VAR
	pGCodeTool		: POINTER TO FB_GCodeTool;
END_VAR
CASE eType OF
	E_PrintParamType.Pressure:
		CASE nNumerator OF
			1:	IF aiDispenser[1] <> 0 AND_THEN 
					(aiDispenser[1].P_pObject^.P_eObjectType = E_ObjectType.OBJECTTYPE_CartDispenser OR	aiDispenser[1].P_pObject^.P_eObjectType = E_ObjectType.OBJECTTYPE_CartDispStirrer) THEN
					pGCodeTool := aiDispenser[1].P_pObject;
					M_SetPrintParams := pGCodeTool^.M_SetPrintParams(E_PrintParamType.Pressure, 1, nValue);
				ELSE
					M_SetPrintParams.bError := TRUE;
					M_SetPrintParams.nErrorId := E_ErrorIdCmd.ERRORID_InvalidPrintParamType;
				END_IF
				
			2:	IF aiDispenser[2] <> 0 AND_THEN
					(aiDispenser[2].P_pObject^.P_eObjectType = E_ObjectType.OBJECTTYPE_CartDispenser OR aiDispenser[2].P_pObject^.P_eObjectType = E_ObjectType.OBJECTTYPE_CartDispStirrer) THEN
					pGCodeTool := aiDispenser[2].P_pObject;
					M_SetPrintParams := pGCodeTool^.M_SetPrintParams(E_PrintParamType.Pressure, 1, nValue);
				ELSE
					M_SetPrintParams.bError := TRUE;
					M_SetPrintParams.nErrorId := E_ErrorIdCmd.ERRORID_InvalidPrintParamType;
				END_IF
			
			3: IF aiDispenser[3] <> 0 AND_THEN
					(aiDispenser[3].P_pObject^.P_eObjectType = E_ObjectType.OBJECTTYPE_CartDispenser OR aiDispenser[3].P_pObject^.P_eObjectType = E_ObjectType.OBJECTTYPE_CartDispStirrer) THEN
					pGCodeTool := aiDispenser[3].P_pObject;
					M_SetPrintParams := pGCodeTool^.M_SetPrintParams(E_PrintParamType.Pressure, 1, nValue);
				ELSE
					M_SetPrintParams.bError := TRUE;
					M_SetPrintParams.nErrorId := E_ErrorIdCmd.ERRORID_InvalidPrintParamType;
				END_IF
		ELSE
			M_SetPrintParams.bError := TRUE;
			M_SetPrintParams.nErrorId := E_ErrorIdCmd.ERRORID_InvalidPrintParamNumerator;
		END_CASE
		
	E_PrintParamType.Feed:
		CASE nNumerator OF
			1:	IF aiDispenser[1] <> 0 AND_THEN aiDispenser[1].P_pObject^.P_eObjectType = E_ObjectType.OBJECTTYPE_Extruder THEN
					pGCodeTool := aiDispenser[1].P_pObject;
					M_SetPrintParams := pGCodeTool^.M_SetPrintParams(E_PrintParamType.Feed, 1, nValue);
				ELSE
					M_SetPrintParams.bError := TRUE;
					M_SetPrintParams.nErrorId := E_ErrorIdCmd.ERRORID_InvalidPrintParamType;
				END_IF
			
			2:	IF aiDispenser[2] <> 0 AND_THEN aiDispenser[2].P_pObject^.P_eObjectType = E_ObjectType.OBJECTTYPE_Extruder THEN
					pGCodeTool := aiDispenser[2].P_pObject;
					M_SetPrintParams := pGCodeTool^.M_SetPrintParams(E_PrintParamType.Feed, 1, nValue);
				ELSE
					M_SetPrintParams.bError := TRUE;
					M_SetPrintParams.nErrorId := E_ErrorIdCmd.ERRORID_InvalidPrintParamType;
				END_IF
			
			3:	IF aiDispenser[3] <> 0 AND_THEN aiDispenser[3].P_pObject^.P_eObjectType = E_ObjectType.OBJECTTYPE_Extruder THEN
					pGCodeTool := aiDispenser[3].P_pObject;
					M_SetPrintParams := pGCodeTool^.M_SetPrintParams(E_PrintParamType.Feed, 1, nValue);			
				ELSE
					M_SetPrintParams.bError := TRUE;
					M_SetPrintParams.nErrorId := E_ErrorIdCmd.ERRORID_InvalidPrintParamType;
				END_IF
			
		ELSE
			M_SetPrintParams.bError := TRUE;
			M_SetPrintParams.nErrorId := E_ErrorIdCmd.ERRORID_InvalidPrintParamNumerator;
		END_CASE
		
	E_PrintParamType.Flow:
		CASE nNumerator OF
			1:	IF aiDispenser[1] <> 0 AND_THEN aiDispenser[1].P_pObject^.P_eObjectType = E_ObjectType.OBJECTTYPE_PassivPip THEN
					pGCodeTool := aiDispenser[1].P_pObject;
					M_SetPrintParams := pGCodeTool^.M_SetPrintParams(E_PrintParamType.Flow, 1, nValue);			
				ELSE
					M_SetPrintParams.bError := TRUE;
					M_SetPrintParams.nErrorId := E_ErrorIdCmd.ERRORID_InvalidPrintParamType;
				END_IF
			
			2:	IF aiDispenser[2] <> 0 AND_THEN aiDispenser[2].P_pObject^.P_eObjectType = E_ObjectType.OBJECTTYPE_PassivPip THEN
					pGCodeTool := aiDispenser[2].P_pObject;
					M_SetPrintParams := pGCodeTool^.M_SetPrintParams(E_PrintParamType.Flow, 1, nValue);			
				ELSE
					M_SetPrintParams.bError := TRUE;
					M_SetPrintParams.nErrorId := E_ErrorIdCmd.ERRORID_InvalidPrintParamType;
				END_IF
			
			3:	IF aiDispenser[3] <> 0 AND_THEN aiDispenser[3].P_pObject^.P_eObjectType = E_ObjectType.OBJECTTYPE_PassivPip THEN
					pGCodeTool := aiDispenser[3].P_pObject;
					M_SetPrintParams := pGCodeTool^.M_SetPrintParams(E_PrintParamType.Flow, 1, nValue);
				ELSE
					M_SetPrintParams.bError := TRUE;
					M_SetPrintParams.nErrorId := E_ErrorIdCmd.ERRORID_InvalidPrintParamType;
				END_IF
		ELSE
			M_SetPrintParams.bError := TRUE;
			M_SetPrintParams.nErrorId := E_ErrorIdCmd.ERRORID_InvalidPrintParamNumerator;
		END_CASE
	
ELSE
	M_SetPrintParams.bError := TRUE;
	M_SetPrintParams.nErrorId := E_ErrorIdCmd.ERRORID_InvalidPrintParamType;	
END_CASE
END_METHOD

METHOD M_ToolIsOnMasterSlot : BOOL
VAR_INPUT
	pTool : POINTER TO FB_MzTool;
END_VAR
IF aiDispenser[nMasterSlotNr] <> 0 THEN
	M_ToolIsOnMasterSlot := aiDispenser[nMasterSlotNr].P_pObject = pTool;
END_IF
END_METHOD

PROPERTY P_bSensorMounted : BOOL
GET
VAR
	i : USINT;
	pTool : POINTER TO FB_MzTool;
END_VAR
FOR i := 1 TO 3 BY 1 DO
	IF aiDispenser[i] <> 0 THEN
		pTool := aiDispenser[i].P_pObject;
		IF pTool^.P_bSensorMounted THEN
			P_bSensorMounted := TRUE;
			RETURN;
		END_IF
	END_IF
END_FOR
END_GET
END_PROPERTY

PROPERTY P_eDispenserState : E_DispenserState
GET
IF bBasicDispense THEN
	//falls ein Dispenser in Preparing ist, dann bleibt es auch so
	P_eDispenserState := E_DispenserState.Dispensing;
END_IF
END_GET
END_PROPERTY

PROPERTY P_pMasterTool : POINTER TO FB_MzTool
GET
P_pMasterTool := aiDispenser[nMasterSlotNr].P_pObject;
END_GET
END_PROPERTY

PROPERTY P_stAbsPosPhys : ST_3DPoint
GET
VAR
	pMzTool : POINTER TO FB_MzTool;
END_VAR
IF aiDispenser[nMasterSlotNr] <> 0 THEN
	pMzTool := aiDispenser[nMasterSlotNr].P_pObject;
	P_stAbsPosPhys := pMzTool^.P_stAbsPosPhys;
ELSE
	P_stAbsPosPhys := SUPER^.P_stAbsPosPhys;
END_IF
END_GET
END_PROPERTY

END_FUNCTION_BLOCK

// ---- Objects/Tools/FB_Extruder.TcPOU
FUNCTION_BLOCK FB_Extruder EXTENDS FB_GCodeTool Implements I_Dispenser
VAR_OUTPUT
END_VAR
VAR
	
	//Specproperties

	eExtruderType				: E_ExtruderType;
	
	pFbHeaterRef				: POINTER TO FB_MZHeaterRef;
	pFbExtruderRef				: POINTER TO FB_ExtruderRef;
	pFbExtruderControl			: POINTER TO FB_ExtruderControl;
	
	fbPistonExtruderControl		: FB_PistonExtruderControl;
	fbEndlessExtruderControl_1		: FB_EndlessExtruderTMCM_Control;	//FDM2
	fbEndlessExtruderControl_2		: FB_EndlessExtruderTMCM_Control;	//Screwextruder Uli
	fbEndlessExtruderControl_PD1	: FB_EndlessExtruderTMCM_Control;	//PureDyne_1 Extruder
	fbEndlessExtruderControl_PD2	: FB_EndlessExtruderTMCM_Control;	//PureDyne_2 Extruder
	fbEndlessExtruderControl_PD3	: FB_EndlessExtruderTMCM_Control;	//PureDyne_3 Extruder
	
	fbFDM_EL2521Control			: FB_FDM_EL2521_Control;
	
	nSpecInstanceNr				: USINT;
	
	//****************************************Aktionsvariablen****************************************************
	//Action: "InitTool"
	bInitTool			: BOOL;
	nStateA_InitTool	: USINT;	
	
	//Action: "Extrude"
	bExtrude			: BOOL;
	nStateA_Extrude		: USINT;
	bExtrudeStart		: BOOL;
	
	//Action: "MovePlunger"
	bMovePlunger		: BOOL;
	nStateA_MovePlunger : USINT;
	nMovePlungerPos		: DINT;
	
	//Action: "LockUnlock"
	bLockUnlock				: BOOL;
	nStateA_LockUnlock		: USINT;
	nLockUnLockOffset		: DINT;
	
	//Action: "Heating"
	bHeating 			: BOOL;
	nStateA_Heating		: USINT;		//State von A_Heating()
	nTempSetpointCart	: UINT;			//Solltemperatur Kartusche (Temp1)
	nTempSetpointNozzle	: UINT;			//Solltemperatur Nozzle (Temp2)
	nTempSetpointMixer	: UINT;			//Solltemperatur Mixer (Temp3) (nur wenn Master bei TwinExtruder relevant) 
	bHeatingOn			: BOOL;			//Heizung "EIN"

	fbHeaterCtrl		: FB_MzHeaterControl;

	bIsExtruding		: BOOL;
END_VAR

VAR CONSTANT
	cHotTemp			: UINT := 500;	//ab dieser Isttemperatur wird Tool als heiß betrachtet (Interlock)
END_VAR

pFbExtruderControl^(pFbExtruderRef:= pFbExtruderRef);

IF eCurrentState = E_MachineState.MACHINESTATE_Active THEN
	
	IF bInitTool THEN
		A_InitTool();
		IF nStateA_InitTool >= 80 THEN
			IF nStateA_InitTool >= 99 THEN
				bError := TRUE;
			END_IF
			bInitTool := FALSE;
			nStateA_InitTool := 0;
			M_RemoveListEntry(nSearchValue:= E_Action.ACTION_Init);
		END_IF		
	END_IF
	
	IF bHeating THEN	//Heizen
		A_Heating();
		IF nStateA_Heating >= 80 THEN
			IF nStateA_Heating >= 99 THEN
				bError := TRUE;
			END_IF
			bHeating := FALSE;
			nStateA_Heating := 0;
			M_RemoveListEntry(nSearchValue:= E_Action.ACTION_Heating);
		END_IF
	END_IF

	IF bExtrude THEN	//Extrudieren
		A_Extrude();
		IF nStateA_Extrude >= 80 THEN
			IF nStateA_Extrude >= 99 THEN
				bError := TRUE;
			END_IF
			bExtrude := FALSE;
			nStateA_Extrude := 0;
			M_RemoveListEntry(nSearchValue:= E_Action.ACTION_Extrude);
		END_IF
	END_IF
	
	IF bMovePlunger THEN
		A_MovePlunger();
		IF nStateA_MovePlunger >= 80 THEN
			IF nStateA_MovePlunger >= 99 THEN
				bError := TRUE;
			END_IF
			bMovePlunger := FALSE;
			nStateA_MovePlunger := 0;
			M_RemoveListEntry(nSearchValue:= E_Action.ACTION_ExtrMovePlunger);
		END_IF
	END_IF
	
	IF bLockUnlock THEN	//Kolben in Ausgangsstellung fahren
		A_LockUnlock();
		IF nStateA_LockUnlock >= 80 THEN
			IF nStateA_LockUnlock >= 99 THEN
				bError := TRUE;
			END_IF
			bLockUnlock := FALSE;
			nStateA_LockUnlock := 0;
			M_RemoveListEntry(nSearchValue:= E_Action.ACTION_LockUnlock);
		END_IF
	END_IF

END_IF

SUPER^();	//FB_MzTool aufrufen

//Prozessdaten aktualisieren
IF pFbHeaterRef > 0 THEN
	stProcessData.n32Data[7] := BOOL_TO_DINT(pFbHeaterRef^.bHeaterIsOn);
	stProcessData.n32Data[8] := pFbHeaterRef^.nTemp1Actual;
	stProcessData.n32Data[9] := pFbHeaterRef^.nTemp2Actual;
	stProcessData.n32Data[13] := pFbHeaterRef^.nTemp3Actual;
END_IF

IF pFbExtruderRef > 0 THEN
	bIsExtruding := pFbExtruderControl^.bBusy;
	stProcessData.n32Data[10] := BOOL_TO_DINT(bIsExtruding);
	stProcessData.n32Data[11] := BOOL_TO_DINT(pFbExtruderRef^.P_bIsLocked);
	stProcessData.n32Data[12] := pFbExtruderRef^.P_nCurrentPos;
END_IF

aObjProcData[nNotifyId] := stProcessData;

ACTION A_Extrude:
IF nStateA_Extrude = 0 THEN
	IF NOT pFbExtruderControl^.bBusy THEN
		nStateA_Extrude := 80;
	END_IF
ELSIF nStateA_Extrude = 70 THEN
	pFbExtruderControl^.M_HardStop();
	nStateA_Extrude := 71;
ELSIF nStateA_Extrude = 71 THEN
	IF NOT pFbExtruderControl^.bBusy THEN
		nStateA_Extrude := 80;
	END_IF
END_IF

IF pFbExtruderControl^.bError THEN
	stError.ErrorId := pFbExtruderControl^.nErrorId;
	stError.POUState := nStateA_Extrude;
	nStateA_Extrude := 99;
END_IF

//Errorhandling
IF nStateA_Extrude = 99 THEN
	stError.Cmd := E_Action.ACTION_Extrude;
	stError.POU := E_POU.POU_FB_Extruder;
	stError.POUAction := E_POUACT.POUACT_A_Extrude;
	fbErrorList.M_Add(stError);
END_IF
END_ACTION

ACTION A_Heating:
IF nStateA_Heating = 0 THEN
	fbHeaterCtrl(bExecute:= TRUE, nTempZone1:= nTempSetpointCart, nTempZone2:= nTempSetpointNozzle,
				nTempZone3:= nTempSetpointMixer, bHeatingOn:= bHeatingOn, pFbHeaterRef:= pFbHeaterRef);

	IF NOT fbHeaterCtrl.bBusy THEN
		IF fbHeaterCtrl.bError THEN
			stError.ErrorId := fbHeaterCtrl.nErrorId; 
			stError.POUState := nStateA_Heating;
			nStateA_Heating := 99;
		ELSE
			nStateA_Heating := 80;	
		END_IF
		fbHeaterCtrl(bExecute:= FALSE, pFbHeaterRef:= pFbHeaterRef);
	END_IF
ELSIF nStateA_Heating = 70 THEN
	fbHeaterCtrl(bExecute:= FALSE, pFbHeaterRef:= pFbHeaterRef);
	nStateA_Heating := 80;
END_IF

//Errorhandling
IF nStateA_Heating = 99 THEN
	stError.POU := E_POU.POU_FB_Extruder;
	stError.Cmd := E_Action.ACTION_Heating;
	stError.POUAction := E_POUACT.POUACT_A_Heating;
	fbErrorList.M_Add(stError);
END_IF
END_ACTION

ACTION A_InitTool:
IF nStateA_InitTool = 0 THEN
	pFbExtruderControl^.M_Init();
	bInitToolOk := TRUE;
	nStateA_InitTool := 80;
END_IF

CASE nStateA_InitTool OF
	0:	pFbExtruderControl^.M_Init();
		nStateA_InitTool := 1;
	1:	IF NOT pFbExtruderControl^.bBusy THEN
			IF pFbExtruderControl^.bError THEN
				nStateA_InitTool := 99;
			ELSE
				nStateA_InitTool := 80;	
			END_IF
		END_IF
END_CASE
END_ACTION

ACTION A_LockUnlock:
//1. Heizer ausschalten falls unlock
IF nStateA_LockUnlock = 0 THEN
	IF pFbExtruderRef^.P_bIsLocked THEN
		IF pFbHeaterRef > 0 THEN
			IF pFbHeaterRef^.bHeaterIsOn THEN
				nStateA_LockUnlock := 1; //weiter zu Heizung ausschalten
			ELSE
				nStateA_LockUnlock := 2; //weiter zu unlocking
			END_IF
		ELSE
			nStateA_LockUnlock := 2; //weiter zu unlocking
		END_IF
	ELSE
		nStateA_LockUnlock := 3; //weiter zu locking
	END_IF
END_IF

CASE nStateA_LockUnlock OF
	1:	//Heizer ausschalten
		fbHeaterCtrl(bExecute:= TRUE, nTempZone1:= nTempSetpointCart, nTempZone2:= nTempSetpointNozzle, 
					bHeatingOn:= FALSE, pFbHeaterRef:= pFbHeaterRef);
	
		IF NOT fbHeaterCtrl.bBusy THEN
			IF fbHeaterCtrl.bError THEN
				stError.ErrorId := fbHeaterCtrl.nErrorId; 
				stError.POUState := nStateA_Heating;
				nStateA_LockUnlock := 99;
			ELSE
				nStateA_LockUnlock := 2;	
			END_IF
			fbHeaterCtrl(bExecute:= FALSE, pFbHeaterRef:= pFbHeaterRef);
		END_IF

	2:	//unlocking
		fbPistonExtruderControl.M_Unlock(nLockUnLockOffset);
		nStateA_LockUnlock := 10;
		
	3:	//locking
		fbPistonExtruderControl.M_Lock(nLockUnLockOffset);
		nStateA_LockUnlock := 10;
	
	10:	
		IF NOT pFbExtruderControl^.bBusy THEN
			nStateA_LockUnlock := 80;
		END_IF
		
	70:
		pFbExtruderControl^.M_HardStop();
		IF fbHeaterCtrl.bBusy THEN
			fbHeaterCtrl(bExecute:= FALSE, pFbHeaterRef:= pFbHeaterRef);	
		END_IF
		nStateA_LockUnlock := 71;
	
	71:	
		IF NOT pFbExtruderControl^.bBusy THEN
			nStateA_LockUnlock := 80;
		END_IF	
END_CASE

IF pFbExtruderControl^.bError THEN
	stError.ErrorId := pFbExtruderControl^.nErrorId;
	stError.POUState := nStateA_LockUnlock;
	nStateA_LockUnlock := 99;
END_IF
//Errorhandling
IF nStateA_LockUnlock = 99 THEN
	stError.Cmd := E_Action.ACTION_LockUnlock;
	stError.POU := E_POU.POU_FB_Extruder;
	stError.POUAction := E_POUACT.POUACT_A_Reload;
	fbErrorList.M_Add(stError);
END_IF
END_ACTION

ACTION A_MovePlunger:
IF nStateA_MovePlunger = 0 THEN
	IF NOT fbPistonExtruderControl.bBusy THEN
		nStateA_MovePlunger := 80;
	END_IF
ELSIF nStateA_MovePlunger = 70 THEN
	fbPistonExtruderControl.M_HardStop();
	nStateA_MovePlunger := 71;
ELSIF nStateA_MovePlunger = 71 THEN
	IF NOT fbPistonExtruderControl.bBusy THEN
		nStateA_MovePlunger := 80;
	END_IF
END_IF

IF fbPistonExtruderControl.bError THEN
	stError.ErrorId := fbPistonExtruderControl.nErrorId;
	stError.POUState := nStateA_MovePlunger;
	nStateA_MovePlunger := 99;
END_IF

//Errorhandling
IF nStateA_MovePlunger = 99 THEN
	stError.Cmd := E_Action.ACTION_ExtrMovePlunger;
	stError.POU := E_POU.POU_FB_Extruder;
	stError.POUAction := E_POUACT.POUACT_A_MovePlunger;
	fbErrorList.M_Add(stError);
END_IF
END_ACTION

ACTION A_Reset:
//Ist noch eine Aktion aktiv?
IF nStateA_ResetSpec = 0 THEN 
	IF bHeating THEN
		bHeating := FALSE;
		nStateA_Heating := 0;
	END_IF
	
	IF pFbExtruderControl^.bError THEN
		pFbExtruderControl^.M_Reset();
	END_IF
	
	nStateA_ResetSpec := 80;		
END_IF

SUPER^.A_Reset();
END_ACTION

ACTION A_Stop:
IF nStateA_Stop = 0 THEN
	IF bHeating AND nStateA_Heating < 70 THEN
		nStateA_Heating := 70;
	END_IF
	
	IF bExtrude AND nStateA_Extrude < 70 THEN
		nStateA_Extrude := 70;
	END_IF
	
	IF bMovePlunger AND nStateA_MovePlunger < 70 THEN
		nStateA_MovePlunger := 70;
	END_IF
	
	IF bLockUnlock AND nStateA_LockUnlock < 70 THEN
		nStateA_LockUnlock := 70;
	END_IF
	
	nStateA_Stop := 1;
END_IF

SUPER^.A_Stop();
END_ACTION

METHOD FB_init : BOOL
VAR_INPUT
	bInitRetains : BOOL; // if TRUE, the retain variables are initialized (warm start / cold start)
	bInCopyCode : BOOL;  // if TRUE, the instance afterwards gets moved into the copy code (online change)
END_VAR

VAR
	nFirstAdress : PVOID;
	nSelfAdress : PVOID;
END_VAR
nFirstAdress := ADR(afbExtruder[1]);
nSelfAdress := THIS;
{IF hasvalue (RegisterSize, '32')}
nSpecInstanceNr := UDINT_TO_USINT((nSelfAdress - nFirstAdress)/SIZEOF(THIS^) + 1);
{ELSE}
nSpecInstanceNr := ULINT_TO_USINT((nSelfAdress - nFirstAdress)/SIZEOF(THIS^) + 1);
{END_IF}
eObjectType := E_ObjectType.OBJECTTYPE_Extruder;
eObjectGroup := E_ObjectGroup.OBJECTGROUP_MzTool OR E_ObjectGroup.OBJECTGROUP_Device;
END_METHOD

METHOD M_AddChild : ERRORID
VAR_INPUT
	pObject : POINTER TO FB_Object;
	nSlotNr	: UINT;
	nIndex 	: INT;
END_VAR
//Der Extruder kann folgende Objekt-Typen aufnehmen
//Nozzle
IF pObject <> 0 THEN
	IF pObject^.P_eObjectType = E_ObjectType.OBJECTTYPE_Nozzle OR
		pObject^.P_eObjectType = E_ObjectType.OBJECTTYPE_DummyTool THEN
		M_AddChild := SUPER^.M_AddChild(pObject,nSlotNr,nIndex);
	ELSIF pObject^.P_eObjectType = E_ObjectType.OBJECTTYPE_ZSensor THEN
		//Darf nur von Spritzenextruder aufgenommen werden
		IF eExtruderType = E_ExtruderType.SyringeExtruder1 THEN
			M_AddChild := SUPER^.M_AddChild(pObject,nSlotNr,nIndex);
		END_IF
	ELSE
		M_AddChild := E_ErrorIdObjMgmt.ERRORID_InvalidParentObject;
	END_IF
ELSE
	M_AddChild := E_ErrorIdObjMgmt.ERRORID_InvalidParentObject;
END_IF
END_METHOD

METHOD M_CancelAction
VAR_INPUT
	eAction : E_Action;
END_VAR
CASE eAction OF
	E_Action.ACTION_Heating:
		IF bHeating AND nStateA_Heating < 70 THEN
			nStateA_Heating := 70;
		END_IF
	E_Action.ACTION_Extrude:
		IF bExtrude AND nStateA_Extrude < 70 THEN
			nStateA_Extrude := 70;
		END_IF
	E_Action.ACTION_ExtrMovePlunger:
		IF bMovePlunger AND nStateA_MovePlunger < 70 THEN
			nStateA_MovePlunger := 70;
		END_IF
	E_Action.ACTION_LockUnlock:
		IF bLockUnlock AND nStateA_LockUnlock < 70 THEN
			nStateA_LockUnlock := 70;
		END_IF
ELSE
	SUPER^.M_CancelAction(eAction);
END_CASE
END_METHOD

METHOD M_CheckAction : ERRORID
VAR_INPUT
	refActionData 	: REFERENCE TO ST_ActionData;
	pCorrelObject	: POINTER TO FB_Object;
END_VAR
CASE refActionData.eAction OF
	E_Action.ACTION_ActionOnArray,
	E_Action.ACTION_CleanTip,
	E_Action.ACTION_MeasureTool,
	E_Action.ACTION_MoveToTarget,
	E_Action.ACTION_TeachTarget:
		//Nur ausführbar, wenn Extruder nicht Bestandteil von TwinExtruder ist
		IF pParentMzTool^.P_eObjectType = E_ObjectType.OBJECTTYPE_TwinExtruder THEN
			M_CheckAction := E_ErrorIdCmd.ERRORID_InvalidAction;
			RETURN;
		END_IF
	E_Action.ACTION_Extrude:
		RETURN;
ELSE
	M_CheckAction := SUPER^.M_CheckAction(refActionData, pCorrelObject);
END_CASE
END_METHOD

METHOD M_CheckGCodeStart : ERRORID
VAR_INPUT
END_VAR
IF eExtruderType = E_ExtruderType.PistonExtruder1 OR
	eExtruderType = E_ExtruderType.SyringeExtruder1 THEN
	IF NOT P_bIsLocked THEN
		M_CheckGCodeStart := E_ErrorIdCmd.ERRORID_DeviceNotLocked;
	END_IF
END_IF
END_METHOD

METHOD M_CheckProcDataType : BOOL
VAR_INPUT
	eProcDataType : E_ProcDataType;
END_VAR
IF eProcDataType = E_ProcDataType.PROCDATATYPE_Temp1 OR eProcDataType = E_ProcDataType.PROCDATATYPE_Temp2 THEN
	M_CheckProcDataType := TRUE;
END_IF
END_METHOD

METHOD M_CheckProps : ERRORID
VAR_INPUT
END_VAR

VAR
	pHybridDispenser : POINTER TO FB_HybridDispenser;
END_VAR
M_CheckProps := SUPER^.M_CheckProps();
//Nozzle muss zwingend dran wenn:
//Parent ist kein TwinExtruder
//oder
//Parent ist ein HybridDispenser und hängt am MasterSlot

IF pPiece = 0 THEN
	IF pParentMzTool^.P_eObjectType <> E_ObjectType.OBJECTTYPE_TwinExtruder THEN
		IF pParentMzTool^.P_eObjectType = E_ObjectType.OBJECTTYPE_HybridDispenser THEN
			pHybridDispenser := pParentMzTool;
			IF pHybridDispenser^.M_ToolIsOnMasterSlot(THIS) THEN
				M_CheckProps := E_ErrorIdObjMgmt.ERRORID_NoNozzleOnTool;
			END_IF
		END_IF
	END_IF
END_IF
END_METHOD

METHOD M_DispenserPrepare : ERRORID
VAR_INPUT
END_VAR
END_METHOD

METHOD M_DispenserStart : ERRORID
VAR_INPUT
END_VAR
IF NOT (eCurrentState = E_MachineState.MACHINESTATE_Idle OR
	eCurrentState = E_MachineState.MACHINESTATE_Active OR
	eCurrentState = E_MachineState.MACHINESTATE_Ready) THEN
	M_DispenserStart := E_ErrorIdCmd.ERRORID_InvalidState;
	RETURN;
END_IF

IF NOT pFbExtruderRef^.P_bIsLocked THEN
	M_DispenserStart := E_ErrorIdCmd.ERRORID_DeviceNotLocked;
	RETURN;
END_IF

IF pFbExtruderRef^.P_nFeedOrgin = 0 THEN
	M_DispenserStart := E_ErrorIdCmd.ERRORID_InvalidFeed;
	RETURN;	
END_IF

M_DispenserStart := pFbExtruderControl^.M_SetDistance(0);
IF M_DispenserStart > 0 THEN
	RETURN;
END_IF

IF pFbExtruderControl^.bBusy THEN
	M_DispenserStart := E_ErrorIdCmd.ERRORID_BasicActionActive;
	RETURN;
END_IF

pFbExtruderControl^.M_StartStop(TRUE);
bExtrude := TRUE;
fbList.A_AddHeadValue(hList := hList, putValue := E_Action.ACTION_Extrude);
bBusy := TRUE;
eCurrentState := E_MachineState.MACHINESTATE_Active;
END_METHOD

METHOD M_DispenserStop : ERRORID
VAR_INPUT
END_VAR
IF bExtrude THEN
	pFbExtruderControl^.M_StartStop(FALSE);
END_IF
END_METHOD

METHOD M_ExeAction : ERRORID
VAR_INPUT
	refActionData : REFERENCE TO ST_ActionData;	
END_VAR
IF NOT (eCurrentState = E_MachineState.MACHINESTATE_Idle OR
	eCurrentState = E_MachineState.MACHINESTATE_Active OR
	eCurrentState = E_MachineState.MACHINESTATE_Ready) THEN
	M_ExeAction := E_ErrorIdCmd.ERRORID_InvalidState;
	RETURN;
END_IF

//Extruder, die Bestandteil des TwinExtruders sind, dürfen keine MoveActions ausführen
IF refActionData.eAction = E_Action.ACTION_MoveX OR 
		refActionData.eAction = E_Action.ACTION_MoveY OR
		refActionData.eAction = E_Action.ACTION_MoveXY OR
		refActionData.eAction = E_Action.ACTION_Jog THEN
	IF pParentMzTool^.P_eObjectType = E_ObjectType.OBJECTTYPE_TwinExtruder THEN
		M_ExeAction := E_ErrorIdCmd.ERRORID_InvalidAction;
		RETURN;
	END_IF
ELSIF refActionData.eAction = E_Action.ACTION_MoveZ THEN
	IF pParentMzTool^.P_eObjectType = E_ObjectType.OBJECTTYPE_TwinExtruder THEN
		eMoveModeZ := DINT_TO_USINT(refActionData.aParams[1]);
		IF NOT (eMoveModeZ = E_MoveMode.MODE_Free OR eMoveModeZ = E_MoveMode.MODE_Home) THEN
			M_ExeAction := E_ErrorIdCmd.ERRORID_InvalidAction;
			RETURN;			
		END_IF
	END_IF	
END_IF


CASE refActionData.eAction OF
	 
	E_Action.ACTION_Init:
		IF NOT bInitAxis AND NOT bInitTool THEN
			bInitAxis := TRUE;
			bInitTool := TRUE;
			fbList.A_AddHeadValue( hList := hList, putValue := E_Action.ACTION_Init);	//InitBase
			fbList.A_AddHeadValue( hList := hList, putValue := E_Action.ACTION_Init);	//InitSpec
		ELSE
			RETURN;
		END_IF		

	E_Action.ACTION_Heating:
		IF NOT pFbExtruderRef^.P_bIsLocked THEN
			M_ExeAction := E_ErrorIdCmd.ERRORID_DeviceNotLocked;
			RETURN;
		END_IF
		IF nStateA_Heating = 0 THEN
			nTempSetpointCart := DINT_TO_UINT(refActionData.aParams[1]);
			nTempSetpointNozzle := DINT_TO_UINT(refActionData.aParams[3]);
			nTempSetpointMixer := DINT_TO_UINT(refActionData.aParams[4]);
			IF nTempSetpointCart > 2500 THEN
				M_ExeAction := E_ErrorIdCmd.ERRORID_InvalidHeatingTemp;  //Error
				RETURN;
			END_IF

			IF nTempSetpointNozzle > 2500 THEN
				M_ExeAction := E_ErrorIdCmd.ERRORID_InvalidHeatingTemp;  //Error
				RETURN;
			END_IF
			
			IF nTempSetpointMixer > 2500 THEN
				M_ExeAction := E_ErrorIdCmd.ERRORID_InvalidHeatingTemp;  //Error
				RETURN;
			END_IF
			
			bHeatingOn := DINT_TO_BOOL(refActionData.aParams[2]);			
			bHeating := TRUE;
			fbList.A_AddHeadValue(hList := hList, putValue := E_Action.ACTION_Heating);
		ELSE
			RETURN;
		END_IF
		
	E_Action.ACTION_Extrude:
		IF NOT pFbExtruderRef^.P_bIsLocked THEN
			M_ExeAction := E_ErrorIdCmd.ERRORID_DeviceNotLocked;
			RETURN;
		END_IF
		
		//Feed < 0 lässt den Extruder rückwärts laufen(nur für Endlos-Extruder relevant)
		IF pFbExtruderRef^.P_nFeedOrgin = 0 THEN
			M_ExeAction := E_ErrorIdCmd.ERRORID_InvalidFeed;
			RETURN;	
		END_IF
		
		bExtrudeStart := DINT_TO_BOOL(refActionData.aParams[2]);
		IF bExtrude AND NOT bExtrudeStart THEN //Ausschalten
				pFbExtruderControl^.M_StartStop(FALSE);
		ELSIF NOT (bExtrude OR bLockUnlock) AND bExtrudeStart THEN //Einschalten
			M_ExeAction := pFbExtruderControl^.M_SetDistance(refActionData.aParams[1]);
			IF M_ExeAction > 0 THEN
				RETURN;
			END_IF
			pFbExtruderControl^.M_StartStop(TRUE);
			bExtrude := TRUE;
			fbList.A_AddHeadValue(hList := hList, putValue := E_Action.ACTION_Extrude);
		ELSE
			RETURN;	
		END_IF
	E_Action.ACTION_ExtrMovePlunger:
		//Nur für Pistonextruder erlaubt
		IF eExtruderType = E_ExtruderType.PistonExtruder1 OR eExtruderType = E_ExtruderType.SyringeExtruder1 THEN
			IF NOT pFbExtruderRef^.P_bIsLocked THEN
				M_ExeAction := E_ErrorIdCmd.ERRORID_DeviceNotLocked;
				RETURN;
			END_IF
			nMovePlungerPos := refActionData.aParams[1];
			IF nMovePlungerPos >= 0 AND nMovePlungerPos <= fbPistonExtruderControl.P_nMaxPos THEN
				IF NOT (bExtrude OR bLockUnlock OR bMovePlunger) THEN
					fbPistonExtruderControl.M_MovePlunger(nMovePlungerPos);
					bMovePlunger := TRUE;
					fbList.A_AddHeadValue(hList := hList, putValue := E_Action.ACTION_ExtrMovePlunger);
				END_IF
			ELSE
				M_ExeAction := E_ErrorIdCmd.ERRORID_InvalidPlungerPos;
				RETURN;
			END_IF
		ELSE
			M_ExeAction := E_ErrorIdCmd.ERRORID_InvalidAction;
			RETURN;
		END_IF

	E_Action.ACTION_LockUnlock:
		IF refActionData.aParams[1] = 0 AND NOT pFbExtruderRef^.P_bIsLocked THEN
			M_ExeAction := E_ErrorIdCmd.ERRORID_DeviceAlreadyUnLocked;
			RETURN;
		ELSIF refActionData.aParams[1] = 1 AND pFbExtruderRef^.P_bIsLocked THEN
			M_ExeAction := E_ErrorIdCmd.ERRORID_DeviceAlreadyLocked;
			RETURN;
		END_IF
		
		IF NOT (bExtrude OR bLockUnlock OR bMovePlunger) THEN
			nLockUnLockOffset := refActionData.aParams[2];
			bLockUnlock := TRUE;
			fbList.A_AddHeadValue(hList := hList, putValue := E_Action.ACTION_LockUnlock);
		END_IF
	ELSE
		M_ExeAction := SUPER^.M_ExeAction(refActionData);
		RETURN;
END_CASE

bBusy := TRUE;
eCurrentState := E_MachineState.MACHINESTATE_Active;
END_METHOD

METHOD M_GetAllProps : ERRORID
VAR_INPUT
	refCmdData : REFERENCE TO  ST_CmdData;
END_VAR
//Basisproperties lesen
SUPER^.M_GetAllProps(refCmdData);
//Specialproperties lesen
nCurrentPropIndex := nCurrentPropIndex + 1; 
refCmdData.n32Data[nCurrentPropIndex] := eExtruderType;
nCurrentPropIndex := nCurrentPropIndex + 1;
refCmdData.n32Data[nCurrentPropIndex] := REAL_TO_DINT(pFbExtruderRef^.P_rFactorFeed * 1000000.0);
nCurrentPropIndex := nCurrentPropIndex + 1;
refCmdData.n32Data[nCurrentPropIndex] := REAL_TO_DINT(pFbExtruderRef^.P_rFactorDistance * 1000000.0);
nCurrentPropIndex := nCurrentPropIndex + 1;
refCmdData.n32Data[nCurrentPropIndex] := pFbExtruderControl^.P_nFeed;
nCurrentPropIndex := nCurrentPropIndex + 1; 
refCmdData.n32Data[nCurrentPropIndex] := pFbExtruderControl^.P_nCompFeed;
nCurrentPropIndex := nCurrentPropIndex + 1; 
refCmdData.n32Data[nCurrentPropIndex] := pFbExtruderControl^.P_nRelaxFeed;
nCurrentPropIndex := nCurrentPropIndex + 1;
refCmdData.n32Data[nCurrentPropIndex] := pFbExtruderControl^.P_nCompDistance;
nCurrentPropIndex := nCurrentPropIndex + 1;
refCmdData.n32Data[nCurrentPropIndex] := pFbExtruderControl^.P_nRelaxDistance;
nCurrentPropIndex := nCurrentPropIndex + 1;
IF pFbHeaterRef > 0 THEN
	refCmdData.n32Data[nCurrentPropIndex] := BOOL_TO_DINT(pFbHeaterRef^.P_bHeaterFixed);
ELSE
	refCmdData.n32Data[nCurrentPropIndex] := 0;
END_IF
END_METHOD

METHOD M_GetProcData : DINT
VAR_INPUT
	eProcDataType : E_ProcDataType;
END_VAR
IF eProcDataType = E_ProcDataType.PROCDATATYPE_Temp1 THEN
	M_GetProcData := pFbHeaterRef^.nTemp1Actual;
ELSIF eProcDataType = E_ProcDataType.PROCDATATYPE_Temp2 THEN
	M_GetProcData := pFbHeaterRef^.nTemp2Actual;
END_IF
END_METHOD

METHOD M_SetAllProps : ERRORID
VAR_INPUT
	refCmdData : REFERENCE TO  ST_CmdData;
END_VAR

VAR
	pHybridDispenser : POINTER TO FB_HybridDispenser;
END_VAR
M_SetAllProps := SUPER^.M_SetAllProps(refCmdData);

IF M_SetAllProps > 0 THEN
	RETURN;
END_IF

pFbHeaterRef := 0;

//In Abhängigkeit vom SubType setzen
nCurrentPropIndex := nCurrentPropIndex + 1;
nSpecPropIndex := nCurrentPropIndex;
eExtruderType := DINT_TO_USINT(refCmdData.n32Data[nCurrentPropIndex]);
IF eExtruderType = E_ExtruderType.PistonExtruder1 THEN
	//Parent TwinExtruder ?
	IF pParentMzTool^.P_eObjectType = E_ObjectType.OBJECTTYPE_TwinExtruder THEN
		//folgende Möglichkeiten gibt es
		//Zuordnung zur richtigen Z-Achse - wie?
		//ExtruderRef darf nur einmal belegt sein
		IF pParentSlot^.P_nNr = 1 THEN
			//1. ParentSlotNr = 1 -> Antriebs-Achse 7 , ExtruderRef 5 (SlaveExtruder)
			pFbExtruderRef := ADR(pFbMultiZ^.aFbExtruderRef[5]);
			pFbHeaterRef := ADR(pFbMultiZ^.aFbHeaterRef[5]);
			pFbMultiZ^.aFbZAxisRef[5].eFixedToolType := E_MzToolType.TOOL_TYPE_HTExtruder;	
		ELSIF pParentSlot^.P_nNr = 2 THEN
			//2. ParentSlotNr = 2 -> Antriebs-Achse 7 , ExtruderRef 7 (MasterExtruder)
			pFbExtruderRef := ADR(pFbMultiZ^.aFbExtruderRef[7]);
			pFbHeaterRef := ADR(pFbMultiZ^.aFbHeaterRef[7]);
			pFbMultiZ^.aFbZAxisRef[7].eFixedToolType := E_MzToolType.TOOL_TYPE_HTExtruder;
		ELSE
			M_SetAllProps := E_ErrorIdObjMgmt.ERRORID_ExtruderInWrongSlot;
			RETURN;		
		END_IF
	ELSE
		pFbExtruderRef := ADR(pFbMultiZ^.aFbExtruderRef[pZAxisRef^.nChannel]);
		pZAxisRef^.eFixedToolType := E_MzToolType.TOOL_TYPE_HTExtruder;	
		pFbHeaterRef := ADR(pFbMultiZ^.aFbHeaterRef[pZAxisRef^.nChannel]);
	END_IF
	pFbExtruderControl := ADR(fbPistonExtruderControl);
	fbPistonExtruderControl.P_eSubType := E_ExtruderType.PistonExtruder1;
ELSIF eExtruderType = E_ExtruderType.FilamentExtruder1 THEN	//Das ist die alte Variante mit EL2521
	{IF defined(FDM1)}
		pFbExtruderControl := ADR(fbFDM_EL2521Control);
		pFbExtruderRef := ADR(fbFDM_EL2521Ref);
	{ELSE]}
		M_SetAllProps := E_ErrorIdObjMgmt.ERRORID_FDM1_NotDefined;
		RETURN;
	{END_IF}
	pZAxisRef^.eFixedToolType := E_MzToolType.TOOL_TYPE_None;
ELSIF eExtruderType = E_ExtruderType.FilamentExtruder2 THEN	//Variante mit TMCM1140
	{IF defined(FDM2)}
		pFbExtruderControl := ADR(fbEndlessExtruderControl_1);
		pFbExtruderRef := ADR(fbEndlessExtrTMCMRef);
	{ELSE]}
		M_SetAllProps := E_ErrorIdObjMgmt.ERRORID_FDM2_NotDefined;
		RETURN;
	{END_IF}
	pZAxisRef^.eFixedToolType := E_MzToolType.TOOL_TYPE_None;
	
	ELSIF eExtruderType = E_ExtruderType.PureDyne_1 THEN	//Variante mit TMCM1140
	{IF defined(Pure1)}
		pFbExtruderControl := ADR(fbEndlessExtruderControl_PD1);
		pFbExtruderRef := ADR(fbEndlessExtrTMCMRef_Pure1);
	{ELSE]}
		M_SetAllProps := E_ErrorIdObjMgmt.ERRORID_PureDyne1_NotDefined;
		RETURN;
	{END_IF}
	//pZAxisRef^.eFixedToolType := E_MzToolType.TOOL_TYPE_None;	
	
ELSIF eExtruderType = E_ExtruderType.PureDyne_2 THEN	//Variante mit TMCM1140
	{IF defined(Pure2)}
		pFbExtruderControl := ADR(fbEndlessExtruderControl_PD2);
		pFbExtruderRef := ADR(fbEndlessExtrTMCMRef_Pure2);
	{ELSE]}
		M_SetAllProps := E_ErrorIdObjMgmt.ERRORID_PureDyne2_NotDefined;
		RETURN;
	{END_IF}
	//pZAxisRef^.eFixedToolType := E_MzToolType.TOOL_TYPE_None;	
	
ELSIF eExtruderType = E_ExtruderType.PureDyne_3 THEN	//Variante mit TMCM1140
	{IF defined(Pure3)}
		pFbExtruderControl := ADR(fbEndlessExtruderControl_PD3);
		pFbExtruderRef := ADR(fbEndlessExtrTMCMRef_Pure3);
	{ELSE]}
		M_SetAllProps := E_ErrorIdObjMgmt.ERRORID_PureDyne3_NotDefined;
		RETURN;
	{END_IF}
	//pZAxisRef^.eFixedToolType := E_MzToolType.TOOL_TYPE_None;	
	
ELSIF eExtruderType = E_ExtruderType.ScrewExtruder1 THEN
	{IF defined(SCREWEXTR1)}
		pFbExtruderControl := ADR(fbEndlessExtruderControl_2);
		pFbExtruderRef := ADR(fbHwRefScrewExtr_TMCM);
	{ELSE]}
		M_SetAllProps := E_ErrorIdObjMgmt.ERRORID_SCREWEXTR1_NotDefined;
		RETURN;
	{END_IF}
ELSIF eExtruderType = E_ExtruderType.SyringeExtruder1 THEN
	//Wenn Parent ein HybridDispenser, dann ist die ZAxisRef anders
	IF pParentMzTool^.P_eObjectType = E_ObjectType.OBJECTTYPE_HybridDispenser THEN
		pHybridDispenser := pParentMzTool;
		//über die ZAxisRef lässt sich auch die ExtruderRef holen
		IF pZAxisRef = 0 THEN
			M_SetAllProps := E_ErrorIdObjMgmt.ERRORID_InvalidAxisRef;
			RETURN;
		END_IF
		pFbExtruderRef := ADR(pFbMultiZ^.aFbExtruderRef[pZAxisRef^.nChannel]);
		pFbExtruderControl := ADR(fbPistonExtruderControl);
		fbPistonExtruderControl.P_eSubType := E_ExtruderType.SyringeExtruder1;
		pZAxisRef^.eFixedToolType := E_MzToolType.TOOL_TYPE_SyringeExtruder;		
	ELSIF pParentMzTool^.P_eObjectType = E_ObjectType.OBJECTTYPE_TwinExtruder THEN
		//Es gibt 2 Möglichkeiten der Bestückung: Antriebsachse 1 oder 7
		IF pZAxisRef^.nChannel = 1 THEN
			IF pParentSlot^.P_nNr = 1 THEN
				pFbExtruderRef := ADR(pFbMultiZ^.aFbExtruderRef[1]);
				pFbMultiZ^.aFbZAxisRef[1].eFixedToolType := E_MzToolType.TOOL_TYPE_SyringeExtruder;
			ELSIF pParentSlot^.P_nNr = 2 THEN
				pFbExtruderRef := ADR(pFbMultiZ^.aFbExtruderRef[3]);
				pFbMultiZ^.aFbZAxisRef[3].eFixedToolType := E_MzToolType.TOOL_TYPE_SyringeExtruder;
			ELSE
				M_SetAllProps := E_ErrorIdObjMgmt.ERRORID_ExtruderInWrongSlot;
				RETURN;		
			END_IF
		ELSIF pZAxisRef^.nChannel = 7 THEN
			IF pParentSlot^.P_nNr = 1 THEN
				pFbExtruderRef := ADR(pFbMultiZ^.aFbExtruderRef[5]);
				pFbMultiZ^.aFbZAxisRef[5].eFixedToolType := E_MzToolType.TOOL_TYPE_SyringeExtruder;
			ELSIF pParentSlot^.P_nNr = 2 THEN
				pFbExtruderRef := ADR(pFbMultiZ^.aFbExtruderRef[7]);
				pFbMultiZ^.aFbZAxisRef[7].eFixedToolType := E_MzToolType.TOOL_TYPE_SyringeExtruder;
			ELSE
				M_SetAllProps := E_ErrorIdObjMgmt.ERRORID_ExtruderInWrongSlot;
				RETURN;		
			END_IF
		ELSE
			M_SetAllProps := E_ErrorIdObjMgmt.ERRORID_ExtruderInWrongSlot;
			RETURN;		
		END_IF
		pFbExtruderControl := ADR(fbPistonExtruderControl);
		fbPistonExtruderControl.P_eSubType := E_ExtruderType.SyringeExtruder1;
	ELSE
		pFbExtruderRef := ADR(pFbMultiZ^.aFbExtruderRef[pZAxisRef^.nChannel]);
		pFbExtruderControl := ADR(fbPistonExtruderControl);
		fbPistonExtruderControl.P_eSubType := E_ExtruderType.SyringeExtruder1;
		pZAxisRef^.eFixedToolType := E_MzToolType.TOOL_TYPE_SyringeExtruder;		
	END_IF
ELSE
	//Invalid SubType
	M_SetAllProps := E_ErrorIdObjMgmt.ERRORID_InvalidExtruderSubType;
	RETURN;
END_IF

//Einmal aufrufen, damit Zeiger im FB gesetzt wird
pFbExtruderControl^(pFbExtruderRef:= pFbExtruderRef);

//FactorFeed
nCurrentPropIndex := nCurrentPropIndex + 1;
IF refCmdData.n32Data[nCurrentPropIndex] = 0 THEN	//Darf keinesfalls "0" sein!
	M_SetAllProps := E_ErrorIdObjMgmt.ERRORID_InvalidFactorFeed;
	RETURN;
END_IF
pFbExtruderRef^.P_rFactorFeed := DINT_TO_REAL(refCmdData.n32Data[nCurrentPropIndex]) / 1000000.0;

//FactorDistance
nCurrentPropIndex := nCurrentPropIndex + 1;
IF refCmdData.n32Data[nCurrentPropIndex] = 0 THEN	//Darf keinesfalls "0" sein!
	M_SetAllProps := E_ErrorIdObjMgmt.ERRORID_InvalidFactorDistance;
	RETURN;
END_IF
pFbExtruderRef^.P_rFactorDistance := DINT_TO_REAL(refCmdData.n32Data[nCurrentPropIndex]) / 1000000.0;

//Feed
nCurrentPropIndex := nCurrentPropIndex + 1;
M_SetAllProps := pFbExtruderControl^.M_SetFeed(refCmdData.n32Data[nCurrentPropIndex]);
IF M_SetAllProps > 0 THEN
	RETURN;
END_IF

//CompressFeed
nCurrentPropIndex := nCurrentPropIndex + 1;
M_SetAllProps := pFbExtruderControl^.M_SetCompFeed(refCmdData.n32Data[nCurrentPropIndex]);
IF M_SetAllProps > 0 THEN
	RETURN;
END_IF

//RelaxFeed
nCurrentPropIndex := nCurrentPropIndex + 1;
M_SetAllProps := pFbExtruderControl^.M_SetRelaxFeed(refCmdData.n32Data[nCurrentPropIndex]);
IF M_SetAllProps > 0 THEN
	RETURN;
END_IF

//Distance wird in der Action übertragen

//CompressDistance
nCurrentPropIndex := nCurrentPropIndex + 1;
M_SetAllProps := pFbExtruderControl^.M_SetCompDistance(refCmdData.n32Data[nCurrentPropIndex]);
IF M_SetAllProps > 0 THEN
	RETURN;
END_IF

//RelaxDistance
nCurrentPropIndex := nCurrentPropIndex + 1;
M_SetAllProps := pFbExtruderControl^.M_SetRelaxDistance(refCmdData.n32Data[nCurrentPropIndex]);
IF M_SetAllProps > 0 THEN
	RETURN;
END_IF

nCurrentPropIndex := nCurrentPropIndex + 1;

IF pFbHeaterRef > 0 THEN
	pFbHeaterRef^.P_bHeaterFixed := DINT_TO_BOOL(refCmdData.n32Data[nCurrentPropIndex]);	
END_IF

nNoOfProps := nCurrentPropIndex + 1;
END_METHOD

METHOD M_SetFeed : ERRORID
VAR_INPUT
	nValue : UINT;
END_VAR
M_SetFeed := pFbExtruderControl^.M_SetFeed(nValue);
IF M_SetFeed = 0 THEN
	//GUI informieren, dass Parameter geändert wurde
	fbObjectDirectory.M_SetObjChange(nObjectId);
END_IF
END_METHOD

METHOD M_SetPrintParams : ST_MethResult
VAR_INPUT
	eType 		: E_PrintParamType;
	nNumerator	: USINT;
	nValue		: DINT;
END_VAR

VAR
	stActionData : ST_ActionData;
END_VAR
IF eType = E_PrintParamType.Feed THEN
	IF nNumerator <> 1 THEN
		M_SetPrintParams.bError := TRUE;
		M_SetPrintParams.nErrorId := E_ErrorIdCmd.ERRORID_InvalidPrintParamNumerator;
		RETURN;
	END_IF
	M_SetPrintParams.nErrorId := M_SetFeed(DINT_TO_UINT(nValue));
	IF M_SetPrintParams.nErrorId > 0 THEN
		M_SetPrintParams.bError := TRUE;
	ELSE
		fbObjectDirectory.M_SetObjChange(nObjectId);
	END_IF
ELSE
	M_SetPrintParams.bError := TRUE;
	M_SetPrintParams.nErrorId := E_ErrorIdCmd.ERRORID_InvalidPrintParamType;
END_IF
END_METHOD

METHOD M_SetSingleProp : ERRORID
VAR_INPUT
	refCmdData : REFERENCE TO  ST_CmdData;
END_VAR
IF (nSpecPropIndex + 3) = refCmdData.aHeader[1] THEN	//Feed
	M_SetSingleProp := pFbExtruderControl^.M_SetFeed(refCmdData.n32Data[0]);
ELSIF (nSpecPropIndex + 4) = refCmdData.aHeader[1] THEN	//CompressFeed
	M_SetSingleProp := pFbExtruderControl^.M_SetCompFeed(refCmdData.n32Data[0]);
ELSIF (nSpecPropIndex + 5) = refCmdData.aHeader[1] THEN //RelaxFeed
	M_SetSingleProp := pFbExtruderControl^.M_SetRelaxFeed(refCmdData.n32Data[0]);
ELSIF (nSpecPropIndex + 6) = refCmdData.aHeader[1] THEN	//CompressDistance
	M_SetSingleProp := pFbExtruderControl^.M_SetCompDistance(refCmdData.n32Data[0]);
ELSIF (nSpecPropIndex + 7) = refCmdData.aHeader[1] THEN //RelaxDistance
	M_SetSingleProp := pFbExtruderControl^.M_SetRelaxDistance(refCmdData.n32Data[0]);
ELSE
	M_SetSingleProp := SUPER^.M_SetSingleProp(refCmdData);
END_IF
END_METHOD

PROPERTY P_bHasZSensorSlot : BOOL
GET
IF eExtruderType = E_ExtruderType.SyringeExtruder1 THEN
	P_bHasZSensorSlot := TRUE;	
END_IF
END_GET
END_PROPERTY

PROPERTY P_bIsExtruding : BOOL
GET
P_bIsExtruding := bIsExtruding;
END_GET
END_PROPERTY

PROPERTY P_bIsHot : BOOL
GET
IF pFbHeaterRef > 0 THEN
	P_bIsHot := (pFbHeaterRef^.nTemp1Actual >= cHotTemp) OR (pFbHeaterRef^.nTemp2Actual >= cHotTemp);	
END_IF
END_GET
END_PROPERTY

PROPERTY P_bIsLocked : BOOL
GET
P_bIsLocked := pFbExtruderRef^.P_bIsLocked;
END_GET
END_PROPERTY

PROPERTY P_bSensorMounted : BOOL
GET
IF eExtruderType = E_ExtruderType.SyringeExtruder1 THEN
	P_bSensorMounted := pZAxisRef^.stInput.nToolState.1;	
END_IF
END_GET
END_PROPERTY

PROPERTY P_eDispenserState : E_DispenserState
GET
IF bIsExtruding THEN
	P_eDispenserState := E_DispenserState.Dispensing;	
END_IF
END_GET
END_PROPERTY

PROPERTY P_eExtruderType : E_ExtruderType
GET
P_eExtruderType := eExtruderType;
END_GET
END_PROPERTY

END_FUNCTION_BLOCK

// ---- Hardware/MultiZ/Extruder/FB_ExtruderControl.TcPOU
FUNCTION_BLOCK FB_ExtruderControl

VAR_OUTPUT
	bBusy : BOOL;
	bError : BOOL;
	nErrorId : ERRORID;
END_VAR

VAR_IN_OUT
	pFbExtruderRef : POINTER TO FB_ExtruderRef;
END_VAR

VAR
END_VAR

//Basisklasse

METHOD M_HardStop
VAR_INPUT
END_VAR
END_METHOD

METHOD M_Reset
VAR_INPUT
END_VAR
IF bError THEN
	bError := FALSE;
	nErrorId := 0;
END_IF
END_METHOD

METHOD M_SetCompDistance : ERRORID
VAR_INPUT
	nValue : DINT;
END_VAR
END_METHOD

METHOD M_SetCompFeed : ERRORID
VAR_INPUT
	nValue : DINT;
END_VAR
END_METHOD

METHOD M_SetDistance : ERRORID
VAR_INPUT
	nValue : DINT;
END_VAR
END_METHOD

METHOD M_SetFeed : ERRORID
VAR_INPUT
	nValue : DINT;
END_VAR
END_METHOD

METHOD M_SetRelaxDistance : ERRORID
VAR_INPUT
	nValue : DINT;
END_VAR
END_METHOD

METHOD M_Init
VAR_INPUT
END_VAR
END_METHOD

METHOD M_SetRelaxFeed : ERRORID
VAR_INPUT
	nValue : DINT;
END_VAR
END_METHOD

METHOD M_StartStop
VAR_INPUT
	bStart : BOOL;
END_VAR
END_METHOD

PROPERTY P_nCompDistance : DINT
GET
IF pFbExtruderRef > 0 THEN
	P_nCompDistance := pFbExtruderRef^.P_nCompDistanceOrgin;
END_IF
END_GET
END_PROPERTY

PROPERTY P_nCompFeed : DINT
GET
IF pFbExtruderRef > 0 THEN
	P_nCompFeed := pFbExtruderRef^.P_nCompFeedOrgin; 
END_IF
END_GET
END_PROPERTY

PROPERTY P_nDistance : DINT
GET
IF pFbExtruderRef > 0 THEN
	P_nDistance := pFbExtruderRef^.P_nDistanceOrgin; 
END_IF
END_GET
END_PROPERTY

PROPERTY P_nFeed : DINT
GET
IF pFbExtruderRef > 0 THEN
	P_nFeed := pFbExtruderRef^.P_nFeedOrgin; 
END_IF
END_GET
END_PROPERTY

PROPERTY P_nRelaxDistance : DINT
GET
IF pFbExtruderRef > 0 THEN
	P_nRelaxDistance := pFbExtruderRef^.P_nRelaxDistanceOrgin; 
END_IF
END_GET
END_PROPERTY

PROPERTY P_nRelaxFeed : DINT
GET
IF pFbExtruderRef > 0 THEN
	P_nRelaxFeed := pFbExtruderRef^.P_nRelaxFeedOrgin; 
END_IF
END_GET
END_PROPERTY

END_FUNCTION_BLOCK

// ---- Hardware/MultiZ/Extruder/FB_PistonExtruderControl.TcPOU
FUNCTION_BLOCK FB_PistonExtruderControl EXTENDS FB_ExtruderControl

VAR
	eSubType				: E_ExtruderType;
	pFbPistonExtruderRef	: POINTER TO FB_PistonExtruderRef;
	nStateSdo 				: USINT;
	nNextStateSdo			: USINT;
	fbSdoWrite				: FB_SDO_WRITE;
	bSendDistancePending	: BOOL;
	bSendUnlockOffsetPending: BOOL;
	fbList					: FB_LinkedListCtrl;
	hList					: T_HLINKEDLIST;
	aListNodes				: ARRAY[0..6] OF T_LinkedListEntry;
	nListValue				: PVOID;
	
	bLock					: BOOL;
	nLockOffset				: DINT;
	bUnlock					: BOOL;
	nUnlockOffset			: DINT;
	bMovePlunger			: BOOL;
	nMovePos				: DINT;
	nMoveDistance			: DINT;
	nMoveFeed				: DINT;
	bExtrude				: BOOL;
	
	nCompDistanceTemp		: DINT;
	nRelaxDistanceTemp		: DINT;
	nRelaxFeedTemp			: DINT;
	nDistanceTemp			: DINT;
	nFeedTemp				: DINT;
	
	nStateAction			: USINT;
	
	timer					: TON;
	
	bStop					: BOOL;

END_VAR

VAR CONSTANT
	cMaxPosPiston	 		: DINT := 65000;//µm
	cMaxPosSyringe			: DINT := 87000;//µm
	cMaxFeedPiston			: DINT := 3000;//µm/s
	cMaxFeedSyringe			: DINT := 12000;//µm/s
END_VAR

IF pFbExtruderRef = 0 THEN
	RETURN;
END_IF

pFbPistonExtruderRef := pFbExtruderRef;

IF nStateSdo = 0 THEN //nächsten Eintrag aus Liste holen
	fbList.A_GetHead(hList:= hList,getValue=> nListValue);
	IF fbList.bOk THEN
		{IF  hasvalue (RegisterSize, '32')}
		nStateSdo := UDINT_TO_USINT(nListValue);
		{ELSE}
		nStateSdo := ULINT_TO_USINT(nListValue);
		{END_IF}		
		fbList.A_RemoveHeadValue(hList:= hList);
	END_IF
END_IF

IF nStateSdo = 1 THEN	//Feed
	fbSdoWrite(sADSNetID:= pFbPistonExtruderRef^.pMultiZRef^.P_sAdsNetId, nPortNr:= pFbPistonExtruderRef^.pMultiZRef^.P_nAdsPort, 
				nIndex:= cExtruderFeed.nIndex, nSubIndex:= pFbPistonExtruderRef^.nChannel, nDataLength:= cExtruderFeed.nLength,
				nData:= pFbPistonExtruderRef^.P_nFeedCalc, bExecute:= TRUE); 
	
ELSIF nStateSdo = 2 THEN //CompressFeed
	fbSdoWrite(sADSNetID:= pFbPistonExtruderRef^.pMultiZRef^.P_sAdsNetId, nPortNr:= pFbPistonExtruderRef^.pMultiZRef^.P_nAdsPort, 
				nIndex:= cExtruderCompressFeed.nIndex, nSubIndex:= pFbPistonExtruderRef^.nChannel, nDataLength:= cExtruderCompressFeed.nLength,
				nData:= pFbPistonExtruderRef^.P_nCompFeedCalc, bExecute:= TRUE); 
	
ELSIF nStateSdo = 3 THEN //RelaxFeed
	fbSdoWrite(sADSNetID:= pFbPistonExtruderRef^.pMultiZRef^.P_sAdsNetId, nPortNr:= pFbPistonExtruderRef^.pMultiZRef^.P_nAdsPort, 
				nIndex:= cExtruderRelaxFeed.nIndex, nSubIndex:= pFbPistonExtruderRef^.nChannel, nDataLength:= cExtruderRelaxFeed.nLength,
				nData:= pFbPistonExtruderRef^.P_nRelaxFeedCalc, bExecute:= TRUE); 
	
ELSIF nStateSdo = 4 THEN //Distance
	fbSdoWrite(sADSNetID:= pFbPistonExtruderRef^.pMultiZRef^.P_sAdsNetId, nPortNr:= pFbPistonExtruderRef^.pMultiZRef^.P_nAdsPort, 
				nIndex:= cExtruderDistance.nIndex, nSubIndex:= pFbPistonExtruderRef^.nChannel, nDataLength:= cExtruderDistance.nLength,
				nData:= pFbPistonExtruderRef^.P_nDistanceCalc, bExecute:= TRUE);
	
ELSIF nStateSdo = 5 THEN //CompressDistance
	fbSdoWrite(sADSNetID:= pFbPistonExtruderRef^.pMultiZRef^.P_sAdsNetId, nPortNr:= pFbPistonExtruderRef^.pMultiZRef^.P_nAdsPort, 
				nIndex:= cExtruderCompressDistance.nIndex, nSubIndex:= pFbPistonExtruderRef^.nChannel, nDataLength:= cExtruderCompressDistance.nLength,
				nData:= pFbPistonExtruderRef^.P_nCompDistanceCalc, bExecute:= TRUE);

ELSIF nStateSdo = 6 THEN //RelaxDistance
	fbSdoWrite(sADSNetID:= pFbPistonExtruderRef^.pMultiZRef^.P_sAdsNetId, nPortNr:= pFbPistonExtruderRef^.pMultiZRef^.P_nAdsPort, 
				nIndex:= cExtruderRelaxDistance.nIndex, nSubIndex:= pFbPistonExtruderRef^.nChannel, nDataLength:= cExtruderRelaxDistance.nLength,
				nData:= pFbPistonExtruderRef^.P_nRelaxDistanceCalc, bExecute:= TRUE);
				
ELSIF nStateSdo = 7 THEN //UnlockOffset
	fbSdoWrite(sADSNetID:= pFbPistonExtruderRef^.pMultiZRef^.P_sAdsNetId, nPortNr:= pFbPistonExtruderRef^.pMultiZRef^.P_nAdsPort, 
				nIndex:= cExtruderUnlockOffset.nIndex, nSubIndex:= pFbPistonExtruderRef^.nChannel, nDataLength:= cExtruderUnlockOffset.nLength,
				nData:= pFbPistonExtruderRef^.P_nUnlockOffsetCalc, bExecute:= TRUE);				
END_IF

IF NOT fbSdoWrite.bBusy THEN
	IF fbSdoWrite.bError THEN
		bError := TRUE;
		nErrorId := fbSdoWrite.nAdsErrorId;		
	END_IF
	fbSdoWrite(bExecute:= FALSE);
	IF nStateSdo = 4 THEN
		bSendDistancePending := FALSE;
	ELSIF nStateSdo = 7 THEN
		bSendUnlockOffsetPending := FALSE;
	END_IF
	nStateSdo := 0;
END_IF


IF bLock THEN
	A_Lock();
ELSIF bUnlock THEN
	A_Unlock();
ELSIF bMovePlunger THEN
	A_MovePlunger();
ELSIF bExtrude THEN
	A_Extrude();
END_IF

IF nStateAction >= 80 THEN
	IF nStateAction >= 99 THEN
		bError := TRUE;
	END_IF
	bLock := bUnlock := bMovePlunger := bExtrude := FALSE;
	nStateAction := 0;
END_IF

bBusy := bLock OR bUnlock OR bMovePlunger OR bExtrude;

ACTION A_Extrude:
CASE nStateAction OF
	0:	//warten, bis Distance gesendet
		IF NOT bSendDistancePending THEN
			pFbPistonExtruderRef^.pToolCtrl^.0 := TRUE;
			nStateAction := 1;				
		END_IF
		
	1:	//Timeout für active
		timer(IN:=TRUE,PT:=T#1S);
		IF pFbPistonExtruderRef^.P_bIsActive THEN
			timer(IN:=FALSE);
			nStateAction := 2;
		ELSE
			IF timer.Q THEN
				timer(IN:=FALSE);
				nErrorId := E_ErrorIdMultiZ.ERRORID_TimeoutExtrude;
				pFbPistonExtruderRef^.pToolCtrl^ := 0;
				nStateAction := 99;
			END_IF
		END_IF
		
	2:	//warten, bis Extrude fertig
		IF NOT pFbPistonExtruderRef^.P_bIsActive OR bStop THEN
			bStop := FALSE;
			pFbPistonExtruderRef^.pToolCtrl^.0 := FALSE;
			nStateAction := 80;
		END_IF
	
END_CASE
END_ACTION

ACTION A_Lock:
CASE nStateAction OF
	0:	//Wartezyklus
		IF pFbPistonExtruderRef^.P_bIsActive THEN
			nStateAction := 99;
		ELSE
			nStateAction := 1;
		END_IF
	1:	//Locking starten
		pFbPistonExtruderRef^.pToolCtrl^.0 := TRUE;
		pFbPistonExtruderRef^.pToolCtrl^.2 := TRUE;
		//Timeout für active
		timer(IN:=TRUE,PT:=T#1S);
		IF pFbPistonExtruderRef^.P_bIsActive THEN
			pFbPistonExtruderRef^.pToolCtrl^.0 := FALSE;
			timer(IN:=FALSE);
			nStateAction := 2;
		ELSE
			IF timer.Q THEN
				timer(IN:=FALSE);
				nErrorId := E_ErrorIdMultiZ.ERRORID_TimeoutLock;
				nStateAction := 99;
			END_IF
		END_IF
		
	2:	//waiting for "ready state"
		timer(IN:=TRUE,PT:=T#25S);
		IF NOT pFbPistonExtruderRef^.P_bIsActive THEN
			timer(IN:=FALSE);
			IF nLockOffset > 0 AND NOT pFbPistonExtruderRef^.pToolCtrl^.1 THEN
				nStateAction := 3;
			ELSE
				nStateAction := 80;
			END_IF
			pFbPistonExtruderRef^.pToolCtrl^ := 0;
		ELSE
			IF timer.Q THEN
				timer(IN:=FALSE);
				nErrorId := E_ErrorIdMultiZ.ERRORID_TimeoutLock;
				nStateAction := 99;
			END_IF
		END_IF
		
	3:	//auf Offset fahren
		//aktuelle CompDistance, RelaxDistance, Feed, Distance sichern
		nCompDistanceTemp := pFbPistonExtruderRef^.P_nCompDistanceOrgin;
		nRelaxDistanceTemp := pFbPistonExtruderRef^.P_nRelaxDistanceOrgin;
		nFeedTemp := pFbPistonExtruderRef^.P_nFeedOrgin;
		nDistanceTemp := pFbPistonExtruderRef^.P_nDistanceOrgin;
		
		//CompDist + RelaxDist auf 0 setzen
		M_SetCompDistance(0);
		M_SetRelaxDistance(0);
		nMoveFeed := M_SetFeedToMax();
		M_SetDistance(nLockOffset); //Distance auf Offset setzen
		nStateAction := 4;
		
	4:	//warten bis Distance gesendet (andere werden vorher gesendet)
		IF NOT bSendDistancePending THEN
			pFbPistonExtruderRef^.pToolCtrl^.0 := TRUE;
			timer(IN:=FALSE);
			nStateAction := 5;
		END_IF
		
	5:	//waiting for "active state"
		timer(IN:=TRUE,PT:=T#1S);
		IF pFbPistonExtruderRef^.P_bIsActive THEN
			timer(IN:=FALSE);
			//timeout berechnen
			timer.PT := REAL_TO_TIME((DINT_TO_REAL(nLockOffset) / DINT_TO_REAL(nMoveFeed))*10000.0 + 3000.0);
			nStateAction := 6;
		ELSE
			IF timer.Q THEN
				timer(IN:=FALSE);
				nErrorId := E_ErrorIdMultiZ.ERRORID_TimeoutLock;
				nStateAction := 7;
			END_IF
		END_IF
		
	6:	//waiting for "ready state"
		timer(IN:=TRUE);
		IF NOT pFbPistonExtruderRef^.P_bIsActive THEN
			timer(IN:=FALSE);
			pFbPistonExtruderRef^.pToolCtrl^ := 0;
			nStateAction := 7;
		ELSE
			IF timer.Q THEN
				timer(IN:=FALSE);
				nErrorId := E_ErrorIdMultiZ.ERRORID_TimeoutLock;
				nStateAction := 7;
			END_IF
		END_IF
		
	7:	//gesicherte Parameter zurückschreiben
		M_SetCompDistance(nCompDistanceTemp);
		M_SetRelaxDistance(nRelaxDistanceTemp);
		M_SetFeed(nFeedTemp);
		M_SetDistance(nDistanceTemp);
		nStateAction := 8;

	8:	//warten bis Distance gesendet (andere werden vorher gesendet)
		IF NOT bSendDistancePending THEN
			IF nErrorId > 0 THEN
				nStateAction := 99;
			ELSE
				nStateAction := 80;
			END_IF
		END_IF		

END_CASE

IF nStateAction = 99 THEN
	pFbPistonExtruderRef^.pToolCtrl^ := 0;
END_IF
END_ACTION

ACTION A_MovePlunger:
//Ähnlich wie Extrude impl.
//vorher aktuelle Position von Zielposition abziehen
//CompDist und RelaxDist auf 0 setzen
CASE nStateAction OF
	0:	//aktuelle CompDistance, RelaxDistance, Feed, Distance sichern
		nCompDistanceTemp := pFbPistonExtruderRef^.P_nCompDistanceOrgin;
		nRelaxDistanceTemp := pFbPistonExtruderRef^.P_nRelaxDistanceOrgin;
		nRelaxFeedTemp := pFbPistonExtruderRef^.P_nRelaxFeedOrgin;
		nFeedTemp := pFbPistonExtruderRef^.P_nFeedOrgin;
		nDistanceTemp := pFbPistonExtruderRef^.P_nDistanceOrgin;
		
		nStateAction := 1;

		M_SetCompDistance(0);
		IF nMovePos > pFbPistonExtruderRef^.P_nCurrentPos THEN
			M_SetRelaxDistance(0);
			nMoveFeed := M_SetFeedToMax();
			nMoveDistance := nMovePos - pFbPistonExtruderRef^.P_nCurrentPos; 
			M_SetDistance(nMoveDistance);
		ELSIF nMovePos < pFbPistonExtruderRef^.P_nCurrentPos THEN
			nMoveDistance := pFbPistonExtruderRef^.P_nCurrentPos - nMovePos;
			M_SetRelaxDistance(nMoveDistance);
			nMoveFeed := M_SetRelaxFeedToMax();
			M_SetFeedToMax();
			M_SetDistance(1);
		ELSE
			nStateAction := 80;
			RETURN;
		END_IF
		
	1:	//warten bis Distance gesendet (andere werden vorher gesendet)
		IF NOT bSendDistancePending THEN
			pFbPistonExtruderRef^.pToolCtrl^.0 := TRUE;
			nStateAction := 2;
		END_IF
		
	2:	//waiting for "active state"
		timer(IN:=TRUE,PT:=T#1S);
		IF pFbPistonExtruderRef^.P_bIsActive THEN
			timer(IN:=FALSE);
			//timeout berechnen
			timer.PT := REAL_TO_TIME((DINT_TO_REAL(nMoveDistance) / DINT_TO_REAL(nMoveFeed))*10000.0 + 3000.0);
			nStateAction := 3;
		ELSE
			IF timer.Q THEN
				timer(IN:=FALSE);
				nErrorId := E_ErrorIdMultiZ.ERRORID_TimeoutMovePlunger;
				nStateAction := 4;
			END_IF
		END_IF	
		
	3:	//warten, bis Extrude fertig
		timer(IN:=TRUE);
		IF NOT pFbPistonExtruderRef^.P_bIsActive THEN
			timer(IN:=FALSE);
			pFbPistonExtruderRef^.pToolCtrl^ := 0;
			nStateAction := 4;
		ELSE
			IF timer.Q THEN
				timer(IN:=FALSE);
				nErrorId := E_ErrorIdMultiZ.ERRORID_TimeoutMovePlunger;
				nStateAction := 4;
			END_IF
		END_IF
		
	4:	//gesicherte Parameter zurückschreiben
		M_SetCompDistance(nCompDistanceTemp);
		M_SetRelaxDistance(nRelaxDistanceTemp);
		M_SetRelaxFeed(nRelaxFeedTemp);
		M_SetFeed(nFeedTemp);
		M_SetDistance(nDistanceTemp);
		nStateAction := 5;
		
	5:	//warten bis Distance gesendet (andere werden vorher gesendet)
		IF NOT bSendDistancePending THEN
			IF nErrorId > 0 THEN
				nStateAction := 99;
			ELSE
				nStateAction := 80;	
			END_IF
		END_IF			
END_CASE

IF nStateAction = 99 THEN
	pFbPistonExtruderRef^.pToolCtrl^ := 0;
END_IF
END_ACTION

ACTION A_Unlock:
CASE nStateAction OF
	0:	//warten bis nUnlockOffset übertragen
		IF NOT bSendUnlockOffsetPending THEN
			nStateAction := 1;
		END_IF
		
	1:	//UnLocking starten
		pFbPistonExtruderRef^.pToolCtrl^.0 := TRUE;
		pFbPistonExtruderRef^.pToolCtrl^.2 := TRUE;
		//Timeout für active
		timer(IN:=TRUE,PT:=T#1S);
		IF pFbPistonExtruderRef^.P_bIsActive THEN
			pFbPistonExtruderRef^.pToolCtrl^.0 := FALSE;
			timer(IN:=FALSE);
			nStateAction := 2;
		ELSE
			IF timer.Q THEN
				timer(IN:=FALSE);
				nErrorId := E_ErrorIdMultiZ.ERRORID_TimeoutUnLock;
				nStateAction := 99;
			END_IF
		END_IF
		
	2:	//warten, bis UnLocking ready
		timer(IN:=TRUE,PT:=T#70S);
		IF NOT pFbPistonExtruderRef^.P_bIsActive THEN
			timer(IN:=FALSE);
			pFbPistonExtruderRef^.pToolCtrl^ := 0;
			nStateAction := 80;
		ELSE
			IF timer.Q THEN
				timer(IN:=FALSE);
				nErrorId := E_ErrorIdMultiZ.ERRORID_TimeoutUnLock;
				nStateAction := 99;
			END_IF
		END_IF
END_CASE

IF nStateAction = 99 THEN
	pFbPistonExtruderRef^.pToolCtrl^ := 0;
END_IF
END_ACTION

METHOD FB_init : BOOL
VAR_INPUT
	bInitRetains : BOOL; // if TRUE, the retain variables are initialized (warm start / cold start)
	bInCopyCode : BOOL;  // if TRUE, the instance afterwards gets moved into the copy code (online change)
END_VAR
F_CreateLinkedListHnd(ADR(aListNodes ), SIZEOF(aListNodes ), hList);
END_METHOD

METHOD PRIVATE M_Add
VAR_INPUT
	nValue : UDINT;
END_VAR
VAR
	pPosPtr	: POINTER TO T_LinkedListEntry := 0;
END_VAR
//Checken, ob Eintrag schon vorhanden
fbList.A_GetHead(hList:= hList,getValue=> nListValue, getPosPtr=> pPosPtr);
IF fbList.bOk THEN
	IF nValue = nListValue THEN	//Eintrag schon vorhanden
		RETURN;		
	ELSE //Eintrag nicht vorhanden -> weitersuchen
		REPEAT
			fbList.A_GetNext(hList:= hList,getValue=> nListValue, putPosPtr:= pPosPtr, getPosPtr=> pPosPtr);
			IF fbList.bOk THEN
				IF nValue = nListValue THEN	//Eintrag schon vorhanden
					RETURN;
				END_IF
			END_IF
		UNTIL NOT fbList.bOk
		END_REPEAT
	END_IF
END_IF

fbList.A_AddTailValue(hList:= hList, putValue:= nValue);
END_METHOD

METHOD M_HardStop
VAR_INPUT
END_VAR
IF pFbPistonExtruderRef^.P_bIsActive THEN
	pFbPistonExtruderRef^.pToolCtrl^ := 2;
END_IF
END_METHOD

METHOD M_Init
VAR_INPUT
END_VAR

VAR
	i : USINT;
END_VAR
//Alle Parameter übertragen
FOR i := 1 TO 7 BY 1 DO
	M_Add(i);
END_FOR
END_METHOD

METHOD M_Lock
VAR_INPUT
	nOffset : DINT;
END_VAR
IF NOT (pFbPistonExtruderRef^.P_bIsActive OR pFbExtruderRef^.P_bError OR bBusy) THEN
	nLockOffset := nOffset;
	pFbPistonExtruderRef^.pToolCtrl^ := 0;
	bBusy := TRUE;
	bLock := TRUE;	
END_IF
END_METHOD

METHOD M_MovePlunger
VAR_INPUT
	nPosition : DINT;
END_VAR
nMovePos := nPosition;
IF  NOT(pFbPistonExtruderRef^.P_bIsActive OR pFbPistonExtruderRef^.P_bError OR bBusy) THEN
	bBusy := TRUE;
	bMovePlunger := TRUE;
	pFbPistonExtruderRef^.pToolCtrl^ := 0;
END_IF
END_METHOD

METHOD M_SetCompDistance : ERRORID
VAR_INPUT
		nValue : DINT;
END_VAR

VAR
	nMaxCompPos : DINT;
END_VAR
IF eSubType = E_ExtruderType.PistonExtruder1 THEN
	nMaxCompPos  := cMaxPosPiston;
ELSIF eSubType = E_ExtruderType.SyringeExtruder1 THEN
	nMaxCompPos  := cMaxPosSyringe;
ELSE
	M_SetCompDistance := E_ErrorIdObjMgmt.ERRORID_InvalidExtruderSubType;
END_IF

IF nValue >= 0 AND nValue <= nMaxCompPos THEN
	IF pFbPistonExtruderRef > 0 THEN
		IF pFbPistonExtruderRef^.P_nCompDistanceOrgin <> nValue THEN
			pFbPistonExtruderRef^.P_nCompDistanceOrgin := nValue;
			M_Add(5);
		END_IF
	END_IF
ELSE
	M_SetCompDistance := E_ErrorIdObjMgmt.ERRORID_InvalidCompressDistance;
END_IF
END_METHOD

METHOD M_SetCompFeed : ERRORID
VAR_INPUT
	nValue : DINT;
END_VAR

VAR
	nMaxCompFeed : DINT;
END_VAR
IF eSubType = E_ExtruderType.PistonExtruder1 THEN
	nMaxCompFeed := cMaxFeedPiston;
ELSIF eSubType = E_ExtruderType.SyringeExtruder1 THEN
	nMaxCompFeed := cMaxFeedSyringe;
ELSE
	M_SetCompFeed := E_ErrorIdObjMgmt.ERRORID_InvalidExtruderSubType;
END_IF

IF nValue >= 0 AND nValue <= nMaxCompFeed THEN
	IF pFbPistonExtruderRef > 0 THEN
		IF pFbPistonExtruderRef^.P_nCompFeedOrgin <> nValue THEN
			pFbPistonExtruderRef^.P_nCompFeedOrgin := nValue;
			M_Add(2);
		END_IF
	END_IF
ELSE
	M_SetCompFeed := E_ErrorIdObjMgmt.ERRORID_InvalidCompressFeed;
END_IF
END_METHOD

METHOD M_SetDistance : ERRORID
VAR_INPUT
	nValue : DINT;
END_VAR

VAR
	nMaxPos : DINT;
END_VAR
IF eSubType = E_ExtruderType.PistonExtruder1 THEN
	nMaxPos := cMaxPosPiston;
ELSIF eSubType = E_ExtruderType.SyringeExtruder1 THEN
	nMaxPos := cMaxPosSyringe;
ELSE
	M_SetDistance := E_ErrorIdObjMgmt.ERRORID_InvalidExtruderSubType;
END_IF

IF nValue >= 0 AND nValue <= nMaxPos THEN
	IF pFbPistonExtruderRef > 0 THEN
		IF pFbPistonExtruderRef^.P_nDistanceOrgin <> nValue THEN
			pFbPistonExtruderRef^.P_nDistanceOrgin := nValue;
			M_Add(4);
			bSendDistancePending := TRUE;
		END_IF
	END_IF
ELSE
	M_SetDistance := E_ErrorIdObjMgmt.ERRORID_InvalidExtrudeDistance;
END_IF
END_METHOD

METHOD M_SetFeed : ERRORID
VAR_INPUT
	nValue : DINT;
END_VAR

VAR
	nMaxFeed : DINT;
END_VAR
IF eSubType = E_ExtruderType.PistonExtruder1 THEN
	nMaxFeed := cMaxFeedPiston;
ELSIF eSubType = E_ExtruderType.SyringeExtruder1 THEN
	nMaxFeed := cMaxFeedSyringe;
ELSE
	M_SetFeed := E_ErrorIdObjMgmt.ERRORID_InvalidExtruderSubType;
END_IF

IF nValue >= 0 AND nValue <= nMaxFeed THEN
	IF pFbPistonExtruderRef > 0 THEN
		IF pFbPistonExtruderRef^.P_nFeedOrgin <> nValue THEN
			pFbPistonExtruderRef^.P_nFeedOrgin := nValue;
			M_Add(1);
		END_IF
	END_IF
ELSE
	M_SetFeed := E_ErrorIdObjMgmt.ERRORID_InvalidExtrudeFeed;
END_IF
END_METHOD

METHOD M_SetFeedToMax : DINT
VAR_INPUT
END_VAR
IF eSubType = E_ExtruderType.PistonExtruder1 THEN
	M_SetFeed(cMaxFeedPiston);
	M_SetFeedToMax := cMaxFeedPiston;
ELSIF eSubType = E_ExtruderType.SyringeExtruder1 THEN
	M_SetFeed(cMaxFeedSyringe);
	M_SetFeedToMax := cMaxFeedSyringe;
END_IF
END_METHOD

METHOD M_SetRelaxDistance : ERRORID
VAR_INPUT
	nValue : DINT;
END_VAR

VAR
	nMaxRelaxPos : DINT;
END_VAR
IF eSubType = E_ExtruderType.PistonExtruder1 THEN
	nMaxRelaxPos := cMaxPosPiston;
ELSIF eSubType = E_ExtruderType.SyringeExtruder1 THEN
	nMaxRelaxPos := cMaxPosSyringe;
ELSE
	M_SetRelaxDistance := E_ErrorIdObjMgmt.ERRORID_InvalidExtruderSubType;
END_IF

IF nValue >= 0 AND nValue <= nMaxRelaxPos THEN
	IF pFbPistonExtruderRef > 0 THEN
		IF pFbPistonExtruderRef^.P_nRelaxDistanceOrgin <> nValue THEN
			pFbPistonExtruderRef^.P_nRelaxDistanceOrgin := nValue;
			M_Add(6);
		END_IF
	END_IF
ELSE
	M_SetRelaxDistance := E_ErrorIdObjMgmt.ERRORID_InvalidRelaxDistance;
END_IF
END_METHOD

METHOD M_SetRelaxFeed : ERRORID
VAR_INPUT
	nValue : DINT;
END_VAR

VAR
	nMaxRelaxFeed : DINT;
END_VAR
IF eSubType = E_ExtruderType.PistonExtruder1 THEN
	nMaxRelaxFeed := cMaxFeedPiston;
ELSIF eSubType = E_ExtruderType.SyringeExtruder1 THEN
	nMaxRelaxFeed := cMaxFeedSyringe;
ELSE
	M_SetRelaxFeed := E_ErrorIdObjMgmt.ERRORID_InvalidExtruderSubType;
END_IF

IF nValue >= 0 AND nValue <= nMaxRelaxFeed THEN
	IF pFbPistonExtruderRef > 0 THEN
		IF pFbPistonExtruderRef^.P_nRelaxFeedOrgin <> nValue THEN
			pFbPistonExtruderRef^.P_nRelaxFeedOrgin := nValue;
			M_Add(3);
		END_IF
	END_IF
ELSE
	M_SetRelaxFeed := E_ErrorIdObjMgmt.ERRORID_InvalidRelaxFeed;	
END_IF
END_METHOD

METHOD M_SetRelaxFeedToMax : DINT
VAR_INPUT
END_VAR
IF eSubType = E_ExtruderType.PistonExtruder1 THEN
	M_SetRelaxFeed(cMaxFeedPiston);
	M_SetRelaxFeedToMax := cMaxFeedPiston;
ELSIF eSubType = E_ExtruderType.SyringeExtruder1 THEN
	M_SetRelaxFeed(cMaxFeedSyringe);
	M_SetRelaxFeedToMax := cMaxFeedSyringe;
END_IF
END_METHOD

METHOD M_SetUnlockOffset : ERRORID
VAR_INPUT
	nValue : DINT;
END_VAR

VAR
	nMaxUnlockOffset : DINT;
END_VAR
IF eSubType = E_ExtruderType.PistonExtruder1 THEN
	nMaxUnlockOffset := cMaxPosPiston;
ELSIF eSubType = E_ExtruderType.SyringeExtruder1 THEN
	nMaxUnlockOffset := cMaxPosSyringe;
ELSE
	M_SetUnlockOffset := E_ErrorIdObjMgmt.ERRORID_InvalidExtruderSubType;
END_IF

IF nValue >= 0 AND nValue <= nMaxUnlockOffset THEN
	IF pFbPistonExtruderRef > 0 THEN
		IF pFbPistonExtruderRef^.P_nUnlockOffsetOrgin <> nValue THEN
			pFbPistonExtruderRef^.P_nUnlockOffsetOrgin := nValue;
			M_Add(7);
			bSendUnlockOffsetPending := TRUE;
		END_IF
	END_IF
ELSE
	M_SetUnlockOffset := E_ErrorIdObjMgmt.ERRORID_InvalidUnlockOffset;	
END_IF
END_METHOD

METHOD M_StartStop
VAR_INPUT
	bStart : BOOL;
END_VAR
//Extruder darf nur gestartet werden, wenn:
//1. Das Status-bit ist nicht gesetzt
//2. er ist nicht in Error

IF bStart AND NOT (pFbPistonExtruderRef^.P_bIsActive OR pFbPistonExtruderRef^.P_bError OR bBusy) THEN
	bBusy := TRUE;
	bExtrude := TRUE;
	bStop := FALSE;
	pFbPistonExtruderRef^.pToolCtrl^.1 := FALSE; //HardStop
	pFbPistonExtruderRef^.pToolCtrl^.2 := FALSE; //Mode "Lock/Unlock"
ELSE
	bStop := TRUE;
END_IF
END_METHOD

METHOD M_Unlock
VAR_INPUT
	nOffset : DINT;
END_VAR
IF NOT (pFbPistonExtruderRef^.P_bIsActive OR pFbExtruderRef^.P_bError OR bBusy) THEN
	nUnlockOffset := nOffset;
	M_SetUnlockOffset(nUnlockOffset);
	pFbPistonExtruderRef^.pToolCtrl^.2 := FALSE;
	bBusy := TRUE;
	bUnLock := TRUE;
END_IF
END_METHOD

PROPERTY P_eSubType : E_ExtruderType
GET
P_eSubType := eSubType;
END_GET
SET
eSubType := P_eSubType;
END_SET
END_PROPERTY

PROPERTY P_nMaxPos : DINT
GET
IF eSubType = E_ExtruderType.PistonExtruder1 THEN
	P_nMaxPos := cMaxPosPiston;
ELSIF eSubType = E_ExtruderType.SyringeExtruder1 THEN
	P_nMaxPos := cMaxPosSyringe;
END_IF
END_GET
END_PROPERTY

END_FUNCTION_BLOCK

// ---- Hardware/MultiZ/Extruder/FB_EndlessExtruderTMCM_Control.TcPOU
FUNCTION_BLOCK FB_EndlessExtruderTMCM_Control EXTENDS FB_ExtruderControl

VAR
	pEndlessExtruderRef		: POINTER TO FB_EndlessExtruderTMCM_Ref;
	pTMCM1140Ref			: POINTER TO FB_HwRefTMCM1140;
	fbTMCM1140Power			: FB_TMCM1140_Power;
	fbTMCM1140Rotate		: FB_TMCM1140_Rotate;
	fbTMCM1140Move			: FB_TMCM1140_Move;
	
	nState 					: USINT;
	nStateNext 				: USINT;
	
	nStateAction			: USINT;
	
	bCompress				: BOOL;
	bRelax					: BOOL;
	
	bNormalStop				: BOOL;
	bHardStop				: BOOL;
	bCCW					: BOOL;
END_VAR

VAR CONSTANT
	//Diese Einschränkungen sind bei Endlos-Extrudern nicht relevant.
	cMinCompDistance 	: DINT := 0;
	cMaxCompDistance 	: DINT := 500000;
	cMinDistance		: DINT := -100000;
	cMaxDistance 		: DINT := 100000;
	cMinRelaxDistance	: DINT := 0;
	cMaxRelaxDistance 	: DINT := 500000;
	
	cMinCompFeed		: DINT := 0;
	cMaxCompFeed 		: DINT := 48;	//µl/s
	cMinFeed			: DINT := 0;	//µl/s
	cMaxFeed			: DINT := 48;	//µl/s
	cMinRelaxFeed		: DINT := 0;
	cMaxRelaxFeed 		: DINT := 48;	//µl/s
END_VAR

IF pFbExtruderRef = 0 THEN
	RETURN;
END_IF

pEndlessExtruderRef := pFbExtruderRef; //pExtruderRef wird in M_Init der Basisklasse gesetzt
pTMCM1140Ref := pEndlessExtruderRef^.P_pHwRefTMCM1140;

//Workaround für FDM-Fan - Hier gibt es noch die zweite Möglichkeit, es direkt über eine Out von der TMCM zu machen.
IF pEndlessExtruderRef^.P_nTriggerChannel > 0 THEN
	IF pEndlessExtruderRef^.P_eTriggerOutput = E_TriggerOutput.MultiZOutput THEN
		fbMultiZDigiOut.M_On(pEndlessExtruderRef^.P_nTriggerChannel);
	ELSIF pEndlessExtruderRef^.P_eTriggerOutput = E_TriggerOutput.MultiZPWM THEN
 		fbMultiZPWM.M_On(pEndlessExtruderRef^.P_nTriggerChannel, 1000);
	END_IF
END_IF

IF nState = 1 THEN //Compress
	//Bei NormalStop:
	//Compress zu Ende führen und weiter zu Relax
	//Bei HardStop:
	//Compress sofort stoppen dann ready
	bBusy := TRUE;
	IF bCompress THEN
		fbTMCM1140Move(pHwRef:= pTMCM1140Ref, bRelative:= TRUE, nPosition:= pFbExtruderRef^.P_nCompDistanceCalc,
						nSpeed:= pFbExtruderRef^.P_nCompFeedCalc, bStop:= bHardStop, bExecute:= TRUE);
		IF NOT fbTMCM1140Move.bBusy THEN
			IF fbTMCM1140Move.bError THEN
				nErrorId := fbTMCM1140Move.nErrorId;
				nState := 99;
			ELSE
				IF bNormalStop THEN
					nState := 3; //weiter zu Relax
				ELSE
					nState := 2; //weiter zu Extrude	
				END_IF
			END_IF
			fbTMCM1140Move(pHwRef:= pTMCM1140Ref, bExecute:= FALSE);
		END_IF	
	ELSE
		nState := 2; //weiter zu Extrude
	END_IF
END_IF

IF nState = 2 THEN //Extrude
	//Bei NormalStop:
	//Extrude sofort stoppen und weiter zu Relax
	//Bei HardStop:
	//Extrude sofort stoppen dann ready
	A_Extrude();
	IF nStateAction >= 80 THEN
		IF nStateAction >= 99 THEN
			nState := 99;
		ELSE
			IF bHardStop THEN
				nState := 0;
			ELSE
				nState := 3; //weiter zu Relax
			END_IF			
		END_IF
		nStateAction := 0;
	END_IF
END_IF

IF nState = 3 THEN //Relax
	//Bei NormalStop normal zu Ende führen
	//Bei HardStop Relax sofort stoppen
	IF bRelax THEN
		fbTMCM1140Move(pHwRef:= pTMCM1140Ref, bRelative:= TRUE, nPosition:= - pFbExtruderRef^.P_nRelaxDistanceCalc,
						nSpeed:= pFbExtruderRef^.P_nRelaxFeedCalc, bStop:= bHardStop, bExecute:= TRUE);
		IF NOT fbTMCM1140Move.bBusy THEN
			IF fbTMCM1140Move.bError THEN
				nErrorId := fbTMCM1140Move.nErrorId;
				nState := 99;
			ELSE
				nState := 0;
			END_IF
			fbTMCM1140Move(pHwRef:= pTMCM1140Ref, bExecute:= FALSE);
		END_IF	
	ELSE
		nState := 0;
	END_IF	
END_IF

IF nState = 4 THEN //Init
	bBusy := TRUE;
	A_Init();
	IF nStateAction >= 80 THEN
		IF nStateAction >= 99 THEN
			nState := 99;
		ELSE
			nState := 0;	
		END_IF
		nStateAction := 0;
	END_IF
END_IF

IF nState = 5 THEN //Reset
	bBusy := TRUE;
	A_Init();
	IF nStateAction >= 80 THEN
		IF nStateAction >= 99 THEN
			nState := 99;
		ELSE
			nState := 0;
			bError := FALSE;
			nErrorId := 0;
		END_IF
		nStateAction := 0;
	END_IF
END_IF

IF nState = 0 THEN
	bBusy := FALSE;
	IF pEndlessExtruderRef^.P_bError THEN
		nState := 99;
	END_IF
END_IF

IF nState = 99 THEN
	bBusy := FALSE;
	bError := TRUE;
END_IF

ACTION A_Compress:
IF nStateAction = 0 THEN
	fbTMCM1140Move(pHwRef:= pTMCM1140Ref , bRelative:= TRUE, nPosition:= pFbExtruderRef^.P_nCompDistanceCalc,
					nSpeed:= pFbExtruderRef^.P_nCompFeedCalc, bExecute:= TRUE);
	nStateAction := 1;
ELSIF nStateAction = 1 THEN 
	fbTMCM1140Move(pHwRef:= pTMCM1140Ref, bStop:= bNormalStop OR bHardStop);
	IF NOT fbTMCM1140Move.bBusy THEN
		IF fbTMCM1140Move.bError THEN
			nStateAction := 99;
		ELSE
			nStateAction := 80;
		END_IF
		fbTMCM1140Move(pHwRef:= pTMCM1140Ref, bExecute:= FALSE);
	END_IF
END_IF
END_ACTION

ACTION A_Extrude:
IF nStateAction = 0 THEN
	IF bNormalStop THEN
		nStateAction := 80;
		RETURN;
	END_IF
	
	IF pFbExtruderRef^.P_nFeedCalc < 0 THEN
		bCCW := TRUE;
	ELSIF pFbExtruderRef^.P_nFeedCalc > 0 THEN
		bCCW := FALSE;
	ELSE
		nStateAction := 80;
		RETURN;
	END_IF
	
	IF pFbExtruderRef^.P_nDistanceOrgin <> 0 THEN
 		IF bCCW THEN
			fbTMCM1140Move.nPosition := -pFbExtruderRef^.P_nDistanceCalc;
		ELSE
			fbTMCM1140Move.nPosition := pFbExtruderRef^.P_nDistanceCalc;
		END_IF
		fbTMCM1140Move(pHwRef:= pTMCM1140Ref, bRelative:= TRUE, nSpeed:= ABS(pFbExtruderRef^.P_nFeedCalc), bExecute:= TRUE);
		nStateAction := 1;
	ELSE
		fbTMCM1140Rotate(pHwRef:= pTMCM1140Ref, bCCW:= bCCW, nSpeed:= ABS(pFbExtruderRef^.P_nFeedCalc), bExecute:= TRUE);
		nStateAction := 2;
	END_IF
END_IF

IF nStateAction = 1 THEN
	fbTMCM1140Move(pHwRef:= pTMCM1140Ref, bStop:= bNormalStop OR bHardStop);
	IF NOT fbTMCM1140Move.bBusy THEN
		IF fbTMCM1140Move.bError THEN
			nErrorId := fbTMCM1140Move.nErrorId;
			nStateAction := 99;
		ELSE
			nStateAction := 80;	
		END_IF
		fbTMCM1140Move(pHwRef:= pTMCM1140Ref, bExecute:= FALSE);
	END_IF
END_IF

IF nStateAction = 2 THEN
	fbTMCM1140Rotate(pHwRef:= pTMCM1140Ref, bStop:= bNormalStop OR bHardStop);
	IF NOT fbTMCM1140Rotate.bBusy THEN
		IF fbTMCM1140Rotate.bError THEN
			nErrorId := fbTMCM1140Rotate.nErrorId;
			nStateAction := 99;
		ELSE
			nStateAction := 80;	
		END_IF
		fbTMCM1140Rotate(pHwRef:= pTMCM1140Ref, bExecute:= FALSE);
	END_IF	
END_IF
END_ACTION

ACTION A_Init:
IF nStateAction = 0 THEN	//Init
	fbTMCM1140Power(pHwRef:= pTMCM1140Ref, bExecute := TRUE);
	IF NOT fbTMCM1140Power.bBusy THEN
		IF fbTMCM1140Power.bError THEN
			nStateAction := 99;
		ELSE
			nStateAction := 80;
		END_IF
		fbTMCM1140Power(pHwRef:= pTMCM1140Ref, bExecute := FALSE);
	END_IF
END_IF
END_ACTION

ACTION A_Relax:
IF nStateAction = 0 THEN
	fbTMCM1140Move(pHwRef:= pTMCM1140Ref, bRelative:= TRUE, nPosition:= -pFbExtruderRef^.P_nRelaxDistanceCalc,
					nSpeed:= pFbExtruderRef^.P_nRelaxFeedCalc, bExecute:= TRUE);
	nStateAction := 1;
ELSIF nStateAction = 1 THEN
	fbTMCM1140Move(pHwRef:= pTMCM1140Ref, bStop:= bNormalStop OR bHardStop);
	IF NOT fbTMCM1140Move.bBusy THEN
		IF fbTMCM1140Move.bError THEN
			nStateAction := 99;
		ELSE
			nStateAction := 80;	
		END_IF
		fbTMCM1140Move(pHwRef:= pTMCM1140Ref, bExecute:= FALSE);
	END_IF
END_IF
END_ACTION

METHOD M_HardStop
VAR_INPUT
END_VAR
IF bBusy THEN
	bHardStop := TRUE;
END_IF
END_METHOD

METHOD M_Init
VAR_INPUT
END_VAR
nState := 4;
END_METHOD

METHOD M_LockUnlock
VAR_INPUT
END_VAR
END_METHOD

METHOD M_Reset
VAR_INPUT
END_VAR
IF bError THEN
	nState := 5; //Reset
END_IF
END_METHOD

METHOD M_SetCompDistance : ERRORID
VAR_INPUT
	nValue : DINT;	
END_VAR
IF nValue >= 0 THEN
	IF pEndlessExtruderRef > 0 THEN
		IF pEndlessExtruderRef^.P_nCompDistanceOrgin <> nValue THEN
			pEndlessExtruderRef^.P_nCompDistanceOrgin := nValue;
		END_IF
	END_IF
ELSE
	M_SetCompDistance := E_ErrorIdObjMgmt.ERRORID_InvalidCompressDistance;
END_IF
END_METHOD

METHOD M_SetCompFeed : ERRORID
VAR_INPUT
	nValue : DINT;
END_VAR
IF nValue >= 0 THEN
	IF pEndlessExtruderRef > 0 THEN
		IF pEndlessExtruderRef^.P_nCompFeedOrgin <> nValue THEN
			pEndlessExtruderRef^.P_nCompFeedOrgin := nValue;
		END_IF
	END_IF
ELSE
	M_SetCompFeed := E_ErrorIdObjMgmt.ERRORID_InvalidCompressFeed;
END_IF
END_METHOD

METHOD M_SetDistance : ERRORID
VAR_INPUT
	nValue : DINT;
END_VAR
IF nValue >= 0 THEN
	IF pEndlessExtruderRef > 0 THEN
		IF pEndlessExtruderRef^.P_nDistanceOrgin <> nValue THEN
			pEndlessExtruderRef^.P_nDistanceOrgin := nValue;
		END_IF
	END_IF
ELSE
	M_SetDistance := E_ErrorIdObjMgmt.ERRORID_InvalidExtrudeDistance;
END_IF
END_METHOD

METHOD M_SetFeed : ERRORID
VAR_INPUT
	nValue : DINT;
END_VAR
//Feed darf auch negativ sein (rückwärts)
IF nValue <> 0 THEN
	IF pEndlessExtruderRef > 0 THEN
		IF pEndlessExtruderRef^.P_nFeedOrgin <> nValue THEN
			pEndlessExtruderRef^.P_nFeedOrgin := nValue;
		END_IF
	END_IF
ELSE
	M_SetFeed := E_ErrorIdObjMgmt.ERRORID_InvalidExtrudeFeed;
END_IF
END_METHOD

METHOD M_SetRelaxDistance : ERRORID
VAR_INPUT
	nValue : DINT;
END_VAR
IF nValue >= 0 THEN
	IF pEndlessExtruderRef > 0 THEN
		IF pEndlessExtruderRef^.P_nRelaxDistanceOrgin <> nValue THEN
			pEndlessExtruderRef^.P_nRelaxDistanceOrgin := nValue;
		END_IF
	END_IF
ELSE
	M_SetRelaxDistance := E_ErrorIdObjMgmt.ERRORID_InvalidRelaxDistance;
END_IF
END_METHOD

METHOD M_SetRelaxFeed : ERRORID
VAR_INPUT
	nValue : DINT;
END_VAR
IF nValue >= 0 THEN
	IF pEndlessExtruderRef > 0 THEN
		IF pEndlessExtruderRef^.P_nRelaxFeedOrgin <> nValue THEN
			pEndlessExtruderRef^.P_nRelaxFeedOrgin := nValue;
		END_IF
	END_IF
ELSE
	M_SetRelaxFeed := E_ErrorIdObjMgmt.ERRORID_InvalidRelaxFeed;
END_IF
END_METHOD

METHOD M_StartStop
VAR_INPUT
	bStart : BOOL;
END_VAR
IF bStart AND NOT bBusy THEN
	bNormalStop := FALSE;
	bHardStop := FALSE;
	IF pFbExtruderRef^.P_nCompDistanceCalc > 0 AND pFbExtruderRef^.P_nCompFeedCalc > 0 AND pFbExtruderRef^.P_nDistanceCalc >= 0 AND pFbExtruderRef^.P_nFeedCalc > 0 THEN
		bCompress := TRUE;
	ELSE
		bCompress := FALSE;
	END_IF
	IF pFbExtruderRef^.P_nRelaxDistanceCalc > 0 AND pFbExtruderRef^.P_nRelaxFeedCalc > 0 AND pFbExtruderRef^.P_nDistanceCalc >= 0  AND pFbExtruderRef^.P_nFeedCalc > 0 THEN
		bRelax := TRUE;
	ELSE
		bRelax := FALSE;
	END_IF
	nState := 1;
ELSIF NOT bStart AND bBusy THEN
	bNormalStop := TRUE;
END_IF
END_METHOD

END_FUNCTION_BLOCK

// ---- Hardware/MultiZ/Extruder/FB_EndlessExtruderTMCM_Ref.TcPOU
FUNCTION_BLOCK FB_EndlessExtruderTMCM_Ref EXTENDS FB_ExtruderRef
VAR_INPUT
END_VAR
VAR
	pHwRefTMCM1140 	: POINTER TO FB_HwRefTMCM1140;
	eTriggerOutput	: E_TriggerOutput;
	nTriggerChannel	: USINT;	
END_VAR
VAR_OUTPUT
END_VAR

METHOD FB_init : BOOL
VAR_INPUT
	bInitRetains 	: BOOL; // if TRUE, the retain variables are initialized (warm start / cold start)
	bInCopyCode 	: BOOL;  // if TRUE, the instance afterwards gets moved into the copy code (online change)
	pHwRefTMCM1140 	: POINTER TO FB_HwRefTMCM1140;
	//eTriggerOutput	: E_TriggerOutput;
	//nTriggerChannel	: USINT;
END_VAR
THIS^.pHwRefTMCM1140 := pHwRefTMCM1140;
//THIS^.eTriggerOutput := eTriggerOutput;
//THIS^.nTriggerChannel := nTriggerChannel;
END_METHOD

PROPERTY P_bError : BOOL
GET
END_GET
END_PROPERTY

PROPERTY P_bIsActive : BOOL
GET
END_GET
END_PROPERTY

PROPERTY P_bIsLocked : BOOL
GET
P_bIsLocked := TRUE;
END_GET
END_PROPERTY

PROPERTY P_eTriggerOutput : E_TriggerOutput
GET
P_eTriggerOutput := eTriggerOutput;
END_GET
END_PROPERTY

PROPERTY P_nTriggerChannel : USINT
GET
P_nTriggerChannel := nTriggerChannel;
END_GET
END_PROPERTY

PROPERTY P_pHwRefTMCM1140 : POINTER TO FB_HwRefTMCM1140
GET
P_pHwRefTMCM1140 := pHwRefTMCM1140;
END_GET
END_PROPERTY

END_FUNCTION_BLOCK

// ---- Hardware/TMCM-1140/FB_HwRefTMCM1140.TcPOU
FUNCTION_BLOCK FB_HwRefTMCM1140 EXTENDS FB_CanNodeBase
VAR_INPUT
	nControlword	AT%Q* : UINT;
	nMode			AT%Q* : SINT;
	nTargetPosition AT%Q* : DINT;	//PP-mode
	nTargetSpeed	AT%Q* : INT;	//VL-mode (in PP-mode anders Object über SDO)	
END_VAR
VAR_OUTPUT
	nStatusword 	 	AT%I* : UINT;
	nCurrentMode 	 	AT%I* : SINT;
	nDigiInputs 	 	AT%I* : UDINT;
	nCurrentPosIntern 	AT%I* : DINT;
END_VAR

VAR
	//Diese Variablen werden in FB_Init() initialisiert
	bSetDigiOut0		: BOOL;
	bSetDigiOut1		: BOOL;
	nSwitchConfig		: USINT;
	eHomingMethode		: E_TMCM_HomingMethode;
	nMicrostepResol 	: UINT;
	nFullStepRevo		: UINT;     //0-65535
	nRampDivisor		: USINT; 	//0-13 ; erweitert bei PureDyne Anpassung
	nPulseDivisor		: USINT;	//0-13
	
	//////////////////////////////////////////////////
	nStateNext			: USINT;
	bIsHomed 			: BOOL;
	lrMicroStepsPerRevo	: LREAL; //FullstepPerRevo * nMicrostepResol (FB_Init()) 
	nCurrentPosReal		: DINT;
END_VAR

VAR PERSISTENT
	nMaxCurrent				: UINT;	//Maximaler Strom in mA
	nHoldCurrent 			: UINT;	//Haltestrom in mA
	nDistPerMotorRev		: DINT; //Weg der prop Motorumdrehung zurückgelegt wird (hier wird Getriebeübersetzung oder Spindelsteigung
									//mit beachtet) reale Einheit (Weg oder Winkel) 
	nRefPos					: DINT; //reale Einheit (Weg oder Winkel)
	nMinPos					: DINT; //reale Einheit (Weg oder Winkel)
	nMaxPos					: DINT; //reale Einheit (Weg oder Winkel)
	nHomePos				: DINT; //reale Einheit (Weg oder Winkel)
	nFastHomingSpeed		: DINT;	//reale Einheit/s
	nSlowHomingSpeed		: DINT; //reale Einheit/s
	nMaxSpeed				: DINT; //reale Einheit/s

END_VAR

SUPER^();
IF lrMicroStepsPerRevo > 0 THEN
	nCurrentPosReal := LREAL_TO_DINT((DINT_TO_LREAL(nCurrentPosIntern) * nDistPerMotorRev) / lrMicroStepsPerRevo);
END_IF

METHOD FB_init : BOOL
VAR_INPUT
	bInitRetains : BOOL; // if TRUE, the retain variables are initialized (warm start / cold start)
	bInCopyCode  : BOOL;  // if TRUE, the instance afterwards gets moved into the copy code (online change)
	bSetDigiOut0 : BOOL; //bei TMCM-1140 open drain
	bSetDigiOut1 : BOOL; //bei TMCM-1140 5V
	eLimitSwitchLeftConfig 	: E_TMCM_SwitchConfig;
	eLimitSwitchRightConfig : E_TMCM_SwitchConfig;
	eHomeSwitchConfig	: E_TMCM_SwitchConfig;
	eHomingMethode		: E_TMCM_HomingMethode;
	nMicrostepResol 	: UINT; //2, 4, 8, 16, 32, 64, 128 oder 256
	nFullStepRevo		: UINT;  //0-65535
	nRampDivisor		: USINT; //0-13
	nPulseDivisor		: USINT; //0-13
END_VAR

VAR
	nSwitchConfigLimitLeft 	: USINT;
	nSwitchConfigLimitRight : USINT;
	nSwitchConfigHome 		: USINT;
END_VAR
THIS^.bSetDigiOut0 := bSetDigiOut0;
THIS^.bSetDigiOut1 := bSetDigiOut1;
IF eLimitSwitchLeftConfig = E_TMCM_SwitchConfig.Deactivated THEN
	nSwitchConfigLimitLeft := 1;
ELSIF eLimitSwitchLeftConfig = E_TMCM_SwitchConfig.Inverted THEN
	nSwitchConfigLimitLeft := 4;
END_IF
IF eLimitSwitchRightConfig = E_TMCM_SwitchConfig.Deactivated THEN
	nSwitchConfigLimitRight := 2;
ELSIF eLimitSwitchRightConfig = E_TMCM_SwitchConfig.Inverted THEN
	nSwitchConfigLimitRight := 8;
END_IF
IF eHomeSwitchConfig = E_TMCM_SwitchConfig.Deactivated THEN
	nSwitchConfigHome := 16;
ELSIF eHomeSwitchConfig = E_TMCM_SwitchConfig.Inverted THEN
	nSwitchConfigHome := 32;
END_IF
nSwitchConfig := nSwitchConfigLimitLeft OR nSwitchConfigLimitRight OR nSwitchConfigHome;
THIS^.eHomingMethode := eHomingMethode;
THIS^.nMicrostepResol := nMicrostepResol;
THIS^.nFullStepRevo := nFullStepRevo;
THIS^.nRampDivisor := nRampDivisor;
THIS^.nPulseDivisor := nPulseDivisor;
lrMicroStepsPerRevo := nFullStepRevo * nMicrostepResol;
END_METHOD

METHOD M_GetDS402State : E_CoDS402States
VAR_INPUT
END_VAR
IF (nStatusword AND 16#4F) = 0 THEN
	M_GetDS402State := E_CoDS402States.DS402STATE_NotReadyToSwitchOn;
ELSIF (nStatusword AND 16#4F) = 16#40 THEN
	M_GetDS402State := E_CoDS402States.DS402STATE_SwitchOnDisabled;
ELSIF (nStatusword AND 16#6F) = 16#21 THEN
	M_GetDS402State := E_CoDS402States.DS402STATE_ReadyToSwitchOn;
ELSIF (nStatusword AND 16#6F) = 16#23 THEN
	M_GetDS402State := E_CoDS402States.DS402STATE_SwitchedOn;
ELSIF (nStatusword AND 16#6F) = 16#27 THEN
	M_GetDS402State := E_CoDS402States.DS402STATE_OperationEnabled;
ELSIF (nStatusword AND 16#6F) = 16#07 THEN
	M_GetDS402State := E_CoDS402States.DS402STATE_QuickStopActive;
ELSIF (nStatusword AND 16#4F) = 16#0F THEN
	M_GetDS402State := E_CoDS402States.DS402STATE_FaultReactionActive;
ELSIF (nStatusword AND 16#4F) = 16#08 THEN
	M_GetDS402State := E_CoDS402States.DS402STATE_Fault;
ELSE
	M_GetDS402State := E_CoDS402States.DS402STATE_Notspecified;
END_IF
END_METHOD

METHOD M_GetHomingState : E_CoDS402HomingState
VAR_INPUT
END_VAR

VAR 
	nTest : UINT;
END_VAR
//werted nur die Bits 10,12,13 vom Statusword aus
nTest := nStatusword AND 16#3400;
CASE nStatusword AND 16#3400 OF
	16#0000:	M_GetHomingState := E_CoDS402HomingState.HomingInProgress;
	16#0400:	M_GetHomingState := E_CoDS402HomingState.HomingInteruptedOrNotReached;
	16#1000:	M_GetHomingState := E_CoDS402HomingState.HomingAttainedButNotReached;
	16#1400:	M_GetHomingState := E_CoDS402HomingState.HomingSuccess;
	16#2000,
	16#2400		:M_GetHomingState := E_CoDS402HomingState.HomingError;
END_CASE
END_METHOD

METHOD M_RealToInternPos : DINT
VAR_INPUT
	nValue : DINT; //RealPos
END_VAR
//Formel siehe TMCM-Berechungen.xlsx
IF nDistPerMotorRev > 0 THEN //Div/0 vermeiden
	M_RealToInternPos := LREAL_TO_DINT(lrMicroStepsPerRevo * DINT_TO_LREAL(nValue) / nDistPerMotorRev); 
END_IF
END_METHOD

METHOD M_RealToInternSpeed : DINT
VAR_INPUT
	nValue : DINT; //reelle Speed,z.B. µm/s oder °/s. Hängt von Einheit DistancePerRevolution ab
END_VAR

VAR
	lrResult	: LREAL;
END_VAR
//Formel siehe TMCM-Berechungen.xlsx
IF nDistPerMotorRev > 0 THEN //Div/0 vermeiden
	lrResult := (nValue * lrMicroStepsPerRevo * EXPT(2, nPulseDivisor) * 65536) / (nDistPerMotorRev * LREAL#16000000);
	M_RealToInternSpeed := MIN(2047, LREAL_TO_DINT(lrResult));
END_IF
END_METHOD

METHOD M_SetTargetPos : BOOL
VAR_INPUT
	nValue 		: DINT; //Reale Position
	bRelative 	: BOOL;
END_VAR

VAR
	nTempTargetPos : DINT; //Nur für Min/Max Überprüfung
END_VAR
IF bRelative THEN
	nTempTargetPos := nCurrentPosReal + nValue;
ELSE
	nTempTargetPos := nValue;
END_IF

//Wenn MinPos und MaxPos = 0, dann handelt es sich im Antriebe wie FDM-Extruder o.ä.
//Diese haben diese Begrenzung nicht.
IF (nTempTargetPos >= nMinPos) AND (nTempTargetPos <= nMaxPos) OR (nMinPos = 0 AND nMaxPos = 0) THEN
	nTargetPosition := M_RealToInternPos(nValue);
	M_SetTargetPos := TRUE;
END_IF
END_METHOD

METHOD M_SetVLSpeed : BOOL
VAR_INPUT
	nValue 	: DINT; //reelle Speed,z.B. µm/s oder °/s. Hängt von Einheit DistancePerRevolution ab
	bCCW	: BOOL;	//Drehrichtung gehen den Uhrzeigersinn
END_VAR
IF nValue >= 0 AND nValue <= nMaxSpeed THEN
	nTargetSpeed := DINT_TO_INT(M_RealToInternSpeed(nValue));
	IF bCCW THEN
		nTargetSpeed := nTargetSpeed * -1;
	END_IF
	M_SetVLSpeed := TRUE;
END_IF
END_METHOD

PROPERTY P_bHomeSwitch : BOOL
GET
P_bHomeSwitch := nDigiInputs.19;
END_GET
END_PROPERTY

PROPERTY P_bIsHomed : BOOL
GET
P_bIsHomed := bIsHomed;
END_GET
SET
bIsHomed := P_bIsHomed;
END_SET
END_PROPERTY

PROPERTY P_bIsMoving : BOOL
GET
P_bIsMoving := nStatusword.14;
END_GET
END_PROPERTY

PROPERTY P_bLeftLimitSwitch : BOOL
GET
P_bLeftLimitSwitch := nDigiInputs.17;
END_GET
END_PROPERTY

PROPERTY P_bRightLimitSwitch : BOOL
GET
P_bRightLimitSwitch := nDigiInputs.18;
END_GET
END_PROPERTY

PROPERTY P_bSetDigiOut0 : BOOL
GET
P_bSetDigiOut0 := bSetDigiOut0;
END_GET
END_PROPERTY

PROPERTY P_bSetDigiOut1 : BOOL
GET
P_bSetDigiOut1 := bSetDigiOut1;
END_GET
END_PROPERTY

PROPERTY P_eHomingMethode : E_TMCM_HomingMethode
GET
P_eHomingMethode := eHomingMethode;
END_GET
END_PROPERTY

PROPERTY P_nCurrentPosReal : DINT
GET
P_nCurrentPosReal := nCurrentPosReal;
END_GET
END_PROPERTY

PROPERTY P_nDistPerMotorRev : DINT
GET
P_nDistPerMotorRev := nDistPerMotorRev;
END_GET
SET
nDistPerMotorRev := P_nDistPerMotorRev;
fbSettings.M_WritePersData();
END_SET
END_PROPERTY

PROPERTY P_nFastHomingSpeed : DINT
GET
P_nFastHomingSpeed := nFastHomingSpeed;
END_GET
SET
nFastHomingSpeed := P_nFastHomingSpeed;
fbSettings.M_WritePersData();
END_SET
END_PROPERTY

PROPERTY PUBLIC P_nFullStepRevo : UINT
GET
P_nFullStepRevo := nFullStepRevo;
END_GET
END_PROPERTY

PROPERTY P_nHoldCurrent : UINT
GET
P_nHoldCurrent := nHoldCurrent;
END_GET
SET
 nHoldCurrent := P_nHoldCurrent;
 fbSettings.M_WritePersData();
END_SET
END_PROPERTY

PROPERTY P_nHoldCurrentConverted : USINT
GET
VAR
	rValue : REAL;
END_VAR

VAR CONSTANT
	cMaxCurrent : REAL := 2000.0;	//maximaler Strom der Steuerung im mA entspricht 255 
END_VAR
rValue := UINT_TO_REAL(nHoldCurrent);
rValue := 255.0 / cMaxCurrent * rValue;
P_nHoldCurrentConverted := MIN(255,REAL_TO_USINT(rValue));
END_GET
END_PROPERTY

PROPERTY P_nHomePos : DINT
GET
P_nHomePos := nHomePos;
END_GET
SET
nHomePos := P_nHomePos;
fbSettings.M_WritePersData();
END_SET
END_PROPERTY

PROPERTY P_nMaxCurrent : UINT
GET
P_nMaxCurrent := nMaxCurrent;
END_GET
SET
 nMaxCurrent := P_nMaxCurrent;
 fbSettings.M_WritePersData();
END_SET
END_PROPERTY

PROPERTY P_nMaxCurrentConverted : USINT
GET
VAR
	rValue : REAL;
END_VAR

VAR CONSTANT
	cMaxCurrent : REAL := 2000.0;	//maximaler Strom der Steuerung im mA entspricht 255 
END_VAR
rValue := UINT_TO_REAL(nMaxCurrent);
rValue := 255.0 / cMaxCurrent * rValue;
P_nMaxCurrentConverted := MIN(255,REAL_TO_USINT(rValue));
END_GET
END_PROPERTY

PROPERTY P_nMaxPos : DINT
GET
P_nMaxPos := nMaxPos;
END_GET
SET
nMaxPos := P_nMaxPos;
fbSettings.M_WritePersData();
END_SET
END_PROPERTY

PROPERTY P_nMaxSpeed : DINT
GET
P_nMaxSpeed := nMaxSpeed;
END_GET
SET
nMaxSpeed := P_nMaxSpeed;
fbSettings.M_WritePersData();
END_SET
END_PROPERTY

PROPERTY P_nMicrostepResolConverted : USINT
GET
P_nMicrostepResolConverted := LREAL_TO_USINT(LOG(nMicrostepResol)/LOG(2));
END_GET
END_PROPERTY

PROPERTY P_nMinPos : DINT
GET
P_nMinPos := nMinPos;
END_GET
SET
nMinPos := P_nMinPos;
fbSettings.M_WritePersData();
END_SET
END_PROPERTY

PROPERTY P_nPulseDivisor : USINT
GET
P_nPulseDivisor := nPulseDivisor;
END_GET
END_PROPERTY

PROPERTY PUBLIC P_nRampDivisor : USINT
GET
P_nRampDivisor := nRampDivisor;
END_GET
END_PROPERTY

PROPERTY P_nRefPos : DINT
GET
P_nRefPos := nRefPos;
END_GET
SET
nRefPos := P_nRefPos;
fbSettings.M_WritePersData();
END_SET
END_PROPERTY

PROPERTY P_nSlowHomingSpeed : DINT
GET
P_nSlowHomingSpeed := nSlowHomingSpeed;
END_GET
SET
nSlowHomingSpeed := P_nSlowHomingSpeed;
fbSettings.M_WritePersData();
END_SET
END_PROPERTY

PROPERTY P_nSwitchConfig : USINT
GET
P_nSwitchConfig := nSwitchConfig;
END_GET
END_PROPERTY

END_FUNCTION_BLOCK

// ---- Hardware/TMCM-1140/FB_TMCM1140_Power.TcPOU
FUNCTION_BLOCK FB_TMCM1140_Power
VAR_INPUT
	bExecute : BOOL;
END_VAR
VAR_OUTPUT
	bBusy 		: BOOL;
	bError 		: BOOL;
	nErrorId 	: ERRORID;	
END_VAR
VAR_IN_OUT
	pHwRef : POINTER TO FB_HwRefTMCM1140;
END_VAR
VAR
	nState 		: USINT;
	nStateNext 	: USINT;
	fbSdoWrite	: FB_SDO_WRITE;
	nDataDigiOut: DINT;
END_VAR

IF bExecute THEN
	IF nState = 0 THEN
		bBusy := TRUE; 
		CASE pHwRef^.M_GetDS402State() OF
			E_CoDS402States.DS402STATE_Fault:
				pHwRef^.nControlword := 153;	//Reset error
				nState := 1;
			E_CoDS402States.DS402STATE_SwitchOnDisabled:
				nState := 1;
			E_CoDS402States.DS402STATE_ReadyToSwitchOn:
				pHwRef^.nControlword := 0;	//Transition 7 in DS402 statemachine -> geht in Switch on disabled
				nState := 1;
			E_CoDS402States.DS402STATE_SwitchedOn:
				pHwRef^.nControlword := 0;	//Transition 10 in DS402 statemachine -> geht in Switch on disabled
				nState := 1;
			E_CoDS402States.DS402STATE_OperationEnabled:
				pHwRef^.nControlword := 0;	//Shutdown
				nState := 1;
			E_CoDS402States.DS402STATE_NotReadyToSwitchOn:	//Statusword wahrscheinlich nicht gemappt
				nErrorId := E_ErrorIdDS402.ERRORID_NotReadyToSwitchOn;
				nState := 99;
		END_CASE
	END_IF
	
	CASE nState OF
		1:	//Hier sollte noch ein Timeout eingebaut werden?
			IF pHwRef^.M_GetDS402State() = E_CoDS402States.DS402STATE_SwitchOnDisabled THEN
				//max. current
				fbSdoWrite.nIndex := 16#2003;
				fbSdoWrite.nSubIndex := 0;
				fbSdoWrite.nDataLength := 1;
				fbSdoWrite.nData := pHwRef^.P_nMaxCurrentConverted;
				nState := 40;
				nStateNext := 2;
			END_IF
			
		2:	//Hold current
			fbSdoWrite.nIndex := 16#2004;
			fbSdoWrite.nSubIndex := 0;
			fbSdoWrite.nDataLength := 1;
			fbSdoWrite.nData := pHwRef^.P_nHoldCurrentConverted;
			nState := 40;
			nStateNext := 3;

		3:	//Switch parameters (Endlagen)		
			fbSdoWrite.nIndex := 16#2005;
			fbSdoWrite.nSubIndex := 0;
			fbSdoWrite.nDataLength := 4;
			fbSdoWrite.nData := pHwRef^.P_nSwitchConfig;
			nState := 40;
			nStateNext := 4;		
			
		4:	//Brake deaktivieren
			fbSdoWrite.nIndex := 16#200C;
			fbSdoWrite.nSubIndex := 2;
			fbSdoWrite.nDataLength := 1;
			fbSdoWrite.nData := 0;
			nState := 40;
			nStateNext := 5;

		5:	//Position Windows setzen
			fbSdoWrite.nIndex := 16#6067;
			fbSdoWrite.nSubIndex := 0;
			fbSdoWrite.nDataLength := 4;
			fbSdoWrite.nData := 100;
			nState := 40;
			nStateNext := 6;
			
		6:	//Velocity Dimension Index -> Intern (damit die folgenden Werte geschrieben werden können)
			fbSdoWrite.nIndex := 16#208C;
			fbSdoWrite.nSubIndex := 0;
			fbSdoWrite.nDataLength := 1;
			fbSdoWrite.nData := E_TMCM_VeloDim.INTERN;
			nState := 40;
			nStateNext := 7;
			
		7:	//Microstep Resolution
			fbSdoWrite.nIndex := 16#2000;
			fbSdoWrite.nSubIndex := 0;
			fbSdoWrite.nDataLength := 1;
			fbSdoWrite.nData := pHwRef^.P_nMicrostepResolConverted;
			nState := 40;
			nStateNext := 31;
			
		31:	//FullStep Resolution
			fbSdoWrite.nIndex := 16#2001;
			fbSdoWrite.nSubIndex := 0;
			fbSdoWrite.nDataLength := 2;
			fbSdoWrite.nData := pHwRef^.P_nFullStepRevo;
			nState := 40;
			nStateNext := 8;
			
		8:	//Pulse Divisor
			fbSdoWrite.nIndex := 16#2086;
			fbSdoWrite.nSubIndex := 0;
			fbSdoWrite.nDataLength := 1;
			fbSdoWrite.nData := pHwRef^.P_nPulseDivisor;
			nState := 40;
			nStateNext := 9;
			
		9:	//Ramp Divisor
			fbSdoWrite.nIndex := 16#2085;
			fbSdoWrite.nSubIndex := 0;
			fbSdoWrite.nDataLength := 1;
			fbSdoWrite.nData := pHwRef^.P_nRampDivisor;
			nState := 40;
			nStateNext := 10;
			
		10:	//Digital out mask
			fbSdoWrite.nIndex := 16#2703;
			fbSdoWrite.nSubIndex := 2;
			fbSdoWrite.nDataLength := 4;
			nDataDigiOut.16 := pHwRef^.P_bSetDigiOut0;
			nDataDigiOut.17 := pHwRef^.P_bSetDigiOut1;
			fbSdoWrite.nData := nDataDigiOut;
			nState := 40;
			nStateNext := 11;

		11:	//Set digital out
			fbSdoWrite.nIndex := 16#2703;
			fbSdoWrite.nSubIndex := 1;
			fbSdoWrite.nDataLength := 4;
			fbSdoWrite.nData := nDataDigiOut;
			nState := 40;
			nStateNext := 12;
			
		12:	//Change to "Ready to Switched on"
			pHwRef^.nControlword := 6;
			nState := 13;
			
		13:	IF pHwRef^.M_GetDS402State() = E_CoDS402States.DS402STATE_ReadyToSwitchOn THEN
				pHwRef^.nControlword := 7;	//Change to "Switched on"
				nState := 14;
			ELSIF pHwRef^.M_GetDS402State() = E_CoDS402States.DS402STATE_Fault THEN
				nErrorId := E_ErrorIdDS402.ERRORID_FaultState;
				nState := 99;
			END_IF
			
		14:	IF pHwRef^.M_GetDS402State() = E_CoDS402States.DS402STATE_SwitchedOn THEN
				pHwRef^.nControlword := 15;	//Change to "Operation enable"
				nState := 15;
			ELSIF pHwRef^.M_GetDS402State() = E_CoDS402States.DS402STATE_Fault THEN
				nErrorId := E_ErrorIdDS402.ERRORID_FaultState;
				nErrorId := 232;
				nState := 99;
			END_IF
			
		15:	IF pHwRef^.M_GetDS402State() = E_CoDS402States.DS402STATE_OperationEnabled THEN
				nState := 80;
			ELSIF pHwRef^.M_GetDS402State() = E_CoDS402States.DS402STATE_Fault THEN
				nErrorId := E_ErrorIdDS402.ERRORID_FaultState;
				nErrorId := 232;
				nState := 99;
			END_IF
	END_CASE
	
	//Sdo senden
	IF nState = 40 THEN
		fbSdoWrite(sADSNetID:= pHwRef^.P_sAdsNetId, nPortNr:= pHwRef^.P_nAdsPort, bExecute:= TRUE);
		IF NOT fbSdoWrite.bBusy THEN
			IF fbSdoWrite.bError THEN
				nErrorId := fbSdoWrite.nAdsErrorId;
				nState := 99;
			ELSE
				nState := nStateNext;
			END_IF
			fbSdoWrite(bExecute:= FALSE);
		END_IF		
	END_IF
	
	IF nState >= 80 THEN
		bBusy := FALSE;
		IF nState = 99 THEN
			bError := TRUE;
		END_IF
	END_IF

ELSE
	bBusy := FALSE;
	bError := FALSE;
	nErrorId := 0;
	nState := 0;	
END_IF

END_FUNCTION_BLOCK

// ---- Hardware/TMCM-1140/FB_TMCM1140_Rotate.TcPOU
FUNCTION_BLOCK FB_TMCM1140_Rotate
VAR_INPUT
	bExecute	: BOOL;
	bStop		: BOOL;
	bCCW		: BOOL;
	nSpeed		: DINT; //Reale Einheit/s //wenn -1, dann wird ProfileSpeed genommen
END_VAR
VAR_OUTPUT
	bBusy 		: BOOL;
	bError 		: BOOL;
	nErrorId 	: ERRORID;	
END_VAR
VAR_IN_OUT
	pHwRef : POINTER TO FB_HwRefTMCM1140;
END_VAR
VAR
	nState 			: USINT;
	nCurrentSpeed 	: DINT;
	bCurrentCCW		: BOOL;	
END_VAR

IF bExecute THEN
	IF NOT pHwRef^.M_GetDS402State() = E_CoDS402States.DS402STATE_OperationEnabled THEN
		nErrorID := E_ErrorIdDS402.ERRORID_OperationNotEnabled;
		nState := 99;
	END_IF
	
	IF nState = 0 THEN
		bBusy := TRUE;
		
		IF nSpeed = -1 THEN
			nSpeed := pHwRef^.P_nMaxSpeed;
		END_IF
		
		IF NOT pHwRef^.M_SetVLSpeed(nSpeed, bCCW) THEN
			nErrorID := E_ErrorIdHwGeneral.ERRORID_InvalidSpeed;
			nState := 99;
		ELSE
			nCurrentSpeed := nSpeed;
			bCurrentCCW := bCCW;
			pHwRef^.nMode := 2;
			nState := 1;
		END_IF
		
	ELSIF nState = 1 THEN
		IF bStop THEN
			pHwRef^.M_SetVLSpeed(0, FALSE);
			nState := 2;
		ELSE
			IF nSpeed <> nCurrentSpeed OR bCCW <> bCurrentCCW THEN
				IF pHwRef^.M_SetVLSpeed(nSpeed, bCCW) THEN
					nCurrentSpeed := nSpeed;
					bCurrentCCW := bCCW;
				END_IF
			END_IF
			
		END_IF
	ELSIF nState = 2 THEN
		IF NOT pHwRef^.P_bIsMoving THEN
			nState := 80;
		END_IF
	END_IF
	
	IF nState >= 80 THEN
		bBusy := FALSE;
		IF nState = 99 THEN
			bError := TRUE;
		END_IF
	END_IF

ELSE
	bBusy := FALSE;
	bError := FALSE;
	bStop := FALSE;
	nState := 0;	
END_IF

END_FUNCTION_BLOCK

// ---- Hardware/TMCM-1140/FB_TMCM1140_Move.TcPOU
FUNCTION_BLOCK FB_TMCM1140_Move
VAR_INPUT
	bExecute	: BOOL;
	bStop		: BOOL;
	nPosition	: DINT; //Reale Einheit (µm oder 1/10°)
	nSpeed		: DINT; //Reale Einheit/s //wenn -1, dann wird ProfileSpeed genommen
	bRelative	: BOOL;
END_VAR
VAR_OUTPUT
	bBusy 		: BOOL;
	bError 		: BOOL;
	nErrorId 	: ERRORID;	
END_VAR
VAR_IN_OUT
	pHwRef : POINTER TO FB_HwRefTMCM1140;
END_VAR
VAR
	nState 		: USINT;
	fbSdoWrite 	: FB_SDO_WRITE;
END_VAR

IF bExecute THEN
	//Vorbedingungen prüfen
	IF nState = 0 THEN
		bBusy := TRUE;
		(*IF pHwRef^.bError THEN
			nErrorID := E_ErrorIdHWE.HWE_IsInErrorState;
			JMP _Error;
		END_IF
		IF pHWE^.bBusy THEN
			nErrorID := E_ErrorIdHWE.HWE_IsBusy;
			JMP _Error;
		END_IF*)
		
		IF NOT pHwRef^.P_bIsHomed AND NOT bRelative THEN
			nErrorID := E_ErrorIdHwGeneral.ERRORID_DriveNotHomed;
			nState := 99;
		ELSE
			IF nSpeed = -1 THEN
				nSpeed := pHwRef^.P_nMaxSpeed;
			END_IF
			
			IF nSpeed > pHwRef^.P_nMaxSpeed THEN
				nErrorID := E_ErrorIdHwGeneral.ERRORID_InvalidSpeed;
				nState := 99;
			ELSE
				IF NOT pHwRef^.M_SetTargetPos(nPosition, bRelative) THEN
					nErrorID := E_ErrorIdHwGeneral.ERRORID_InvalidPosition;
					nState := 99;
				ELSE
					nState := 1;			
				END_IF
			END_IF			
		END_IF
	END_IF
	
	IF NOT pHwRef^.M_GetDS402State() = E_CoDS402States.DS402STATE_OperationEnabled THEN
		nErrorID := E_ErrorIdDS402.ERRORID_OperationNotEnabled;
		nState := 99;
	END_IF
	
	CASE nState OF
		1:	//Mode auf 1 stellen und PP-Speed schreiben
			pHwRef^.nMode := 1;
			fbSdoWrite(sADSNetID:= pHwRef^.P_sAdsNetId, nPortNr:= pHwRef^.P_nAdsPort,nIndex:= 16#6081, nSubIndex:= 0,
						nDataLength:= 4, nData:= pHwRef^.M_RealToInternSpeed(nSpeed), bExecute := TRUE);
			IF NOT fbSdoWrite.bBusy THEN
				IF fbSdoWrite.bError THEN
					nErrorID := fbSdoWrite.nAdsErrorId;
					nState := 99;
				ELSE
					IF bStop THEN
						nState := 80;
					ELSE
						pHwRef^.nControlword.4 := TRUE;
						pHwRef^.nControlword.6 := bRelative;
						nState := 2;
					END_IF
				END_IF
				fbSdoWrite(bExecute := FALSE);
			END_IF
			
		2:	//Setpoint ACK?
			IF pHwRef^.nStatusword.12 THEN
				pHwRef^.nControlword.4 := FALSE;
				nState := 3;
			END_IF
			
		3:	//Target reached?
			//Das HALT-Bit von von der TMCM1140 nicht unterstützt.
			//Man kann den Mode auf "0" setzen und dann sollter der Motor auch anhalten
			//allerdingt läuft er aus und stoppt nicht sofort
			IF bStop THEN
				pHwRef^.nMode := 0;
				nState := 80;
			END_IF
			
			IF pHwRef^.nStatusword.10 THEN
				nState := 80;
			END_IF
			
	END_CASE
	
	IF nState >= 80 THEN
		bBusy := FALSE;
		IF nState = 99 THEN
			bError := TRUE;
		END_IF
	END_IF

ELSE
	bBusy := FALSE;
	bError := FALSE;
	bStop := FALSE;
	nState := 0;	
END_IF

END_FUNCTION_BLOCK

// ---- Hardware/MultiZ/Extruder/FB_FDM_EL2521_Control.TcPOU
FUNCTION_BLOCK FB_FDM_EL2521_Control EXTENDS FB_ExtruderControl

VAR
	pFbFilamentExtruderRef	: POINTER TO FB_FDM_EL2521_Ref;
	pPTOStepperRef 			: POINTER TO ST_PTOStepperRef;
	fbPTOStepperRotate 		: FB_PTOStepperRotate;
	fbPTOStepperMoveRel		: FB_PTOStepperMoveRel;
	
	nState 					: USINT;
	nStateNext 				: USINT;
	
	nStateAction			: USINT;
	
	bNormalStop				: BOOL;
	bHardStop				: BOOL;
END_VAR

VAR CONSTANT
	cMinCompDistance 	: DINT := 0;
	cMaxCompDistance 	: DINT := 5000;		//µm
	cMinDistance		: DINT := -100000;	//µm
	cMaxDistance 		: DINT := 100000;	//µm
	cMinRelaxDistance	: DINT := 0;
	cMaxRelaxDistance 	: DINT := 5000;//µm
	
	cMinCompFeed		: DINT := 0;
	cMaxCompFeed 		: DINT := 20000;//µm/s
	cMinFeed			: DINT := 0;
	cMaxFeed			: DINT := 20000;//µm/s
	cMinRelaxFeed		: DINT := 0;
	cMaxRelaxFeed 		: DINT := 20000;//µm/s
END_VAR

IF pFbExtruderRef = 0 THEN
	RETURN;
END_IF

pFbFilamentExtruderRef := pFbExtruderRef;
pPTOStepperRef := pFbFilamentExtruderRef^.P_pPTOStepperRef;

IF nState = 1 THEN //Compress
	bBusy := TRUE;
	IF pFbFilamentExtruderRef^.P_nDistanceOrgin < 0 OR pFbFilamentExtruderRef^.P_nCompDistanceOrgin <= 0 THEN
		nState := 2;
	ELSE
		A_Compress();
		IF nStateAction >= 80 THEN
			nStateAction := 0;
			nState := 2;
			IF bHardStop THEN
				nState := 0;
			END_IF
		END_IF
	END_IF
END_IF

IF nState = 2 THEN //Extrude
	bBusy := TRUE;
	A_Extrude();
	IF nStateAction >= 80 THEN
		nState := 3;
		nStateAction := 0;
		IF bHardStop THEN
			nState := 0;
		END_IF
	END_IF
END_IF

IF nState = 3 THEN //Relax
	IF pFbFilamentExtruderRef^.P_nDistanceOrgin < 0 OR pFbFilamentExtruderRef^.P_nRelaxDistanceOrgin <= 0 THEN
		nState := 0;
	ELSE
		A_Relax();
		IF nStateAction >= 80 THEN
			nStateAction := 0;
			nState := 0;
		END_IF
	END_IF	
END_IF

IF nState = 0 THEN
	bBusy := FALSE;
END_IF

ACTION A_Compress:
IF nStateAction = 0 THEN
	fbPTOStepperMoveRel(bExecute:= TRUE, bStop:= bHardStop, nSteps:= -DINT_TO_INT(pFbExtruderRef^.P_nCompDistanceCalc),
						nSpeed:= DINT_TO_UINT(ABS(pFbExtruderRef^.P_nCompFeedCalc)),pPTOStepperRef:= pPTOStepperRef);
	nStateAction := 1;
ELSIF nStateAction = 1 THEN 
	fbPTOStepperMoveRel(bStop:= bHardStop, pPTOStepperRef:= pPTOStepperRef);
	IF NOT fbPTOStepperMoveRel.bBusy THEN
		fbPTOStepperMoveRel(bExecute:= FALSE, pPTOStepperRef:= pPTOStepperRef);
		nStateAction := 80;
	END_IF
END_IF
END_ACTION

ACTION A_Extrude:
IF nStateAction = 0 THEN
	IF bNormalStop THEN
		nStateAction := 80;
		RETURN;
	END_IF
	IF pFbFilamentExtruderRef^.P_nDistanceOrgin < 0 THEN
		fbPTOStepperMoveRel(bExecute:= TRUE, bStop:= bHardStop, nSteps:= -DINT_TO_INT(pFbExtruderRef^.P_nDistanceCalc),
							nSpeed:= DINT_TO_UINT(ABS(pFbExtruderRef^.P_nFeedCalc)),pPTOStepperRef:= pPTOStepperRef);
		nStateAction := 1;
	ELSIF pFbFilamentExtruderRef^.P_nDistanceOrgin > 0 THEN
		fbPTOStepperMoveRel(bExecute:= TRUE, bStop:= bHardStop, nSteps:= -DINT_TO_INT(pFbExtruderRef^.P_nDistanceCalc),
							nSpeed:= DINT_TO_UINT(ABS(pFbExtruderRef^.P_nFeedCalc)),pPTOStepperRef:= pPTOStepperRef);
		nStateAction := 1;
	ELSE
		IF pFbExtruderRef^.P_nFeedCalc < 0 THEN
			fbPTOStepperRotate(bExecute:= TRUE,	bStop:= bHardStop,	bCCW:= TRUE,
							nSpeed:= DINT_TO_UINT(ABS(pFbExtruderRef^.P_nFeedCalc)), pPTOStepperRef:= pPTOStepperRef);		
		ELSIF pFbExtruderRef^.P_nFeedCalc > 0 THEN
			fbPTOStepperRotate(bExecute:= TRUE,	bStop:= bHardStop,	bCCW:= FALSE,
							nSpeed:= DINT_TO_UINT(ABS(pFbExtruderRef^.P_nFeedCalc)), pPTOStepperRef:= pPTOStepperRef);		
		ELSE
			nStateAction := 80;
			RETURN;
		END_IF
		 nStateAction := 2;
	END_IF
END_IF

IF nStateAction = 1 THEN
	fbPTOStepperMoveRel(bStop:= bNormalStop OR bHardStop, pPTOStepperRef:= pPTOStepperRef);
	IF NOT fbPTOStepperMoveRel.bBusy THEN
		fbPTOStepperMoveRel(bExecute:= FALSE, pPTOStepperRef:= pPTOStepperRef);
		nStateAction := 80;
	END_IF
END_IF

IF nStateAction = 2 THEN
	fbPTOStepperRotate(bExecute:= TRUE,	bStop:= bNormalStop OR bHardStop, pPTOStepperRef:= pPTOStepperRef);
	IF NOT fbPTOStepperRotate.bBusy THEN
		fbPTOStepperRotate(bExecute:= FALSE, pPTOStepperRef:= pPTOStepperRef);
		nStateAction := 80;
	END_IF	
END_IF
END_ACTION

ACTION A_Relax:
IF nStateAction = 0 THEN
	fbPTOStepperMoveRel(bExecute:= TRUE, bStop:= bHardStop, nSteps:= DINT_TO_INT(pFbExtruderRef^.P_nRelaxDistanceCalc),
						nSpeed:= DINT_TO_UINT(ABS(pFbExtruderRef^.P_nRelaxFeedCalc)),pPTOStepperRef:= pPTOStepperRef);
	nStateAction := 1;
ELSIF nStateAction = 1 THEN
	fbPTOStepperMoveRel(bStop:= bHardStop, pPTOStepperRef:= pPTOStepperRef);
	IF NOT fbPTOStepperMoveRel.bBusy THEN
		fbPTOStepperMoveRel(bExecute:= FALSE, pPTOStepperRef:= pPTOStepperRef);
		nStateAction := 80;
	END_IF
END_IF
END_ACTION

METHOD M_HardStop
VAR_INPUT
END_VAR
IF bBusy THEN
	bHardStop := TRUE;
END_IF
END_METHOD

METHOD M_LockUnlock
VAR_INPUT
END_VAR
END_METHOD

METHOD M_SetCompDistance : ERRORID
VAR_INPUT
	nValue : DINT;	
END_VAR
IF nValue >= cMinCompDistance AND nValue <= cMaxCompDistance THEN
	IF pFbFilamentExtruderRef > 0 THEN
		IF pFbFilamentExtruderRef^.P_nCompDistanceOrgin <> nValue THEN
			pFbFilamentExtruderRef^.P_nCompDistanceOrgin := nValue;
		END_IF
	END_IF
ELSE
	M_SetCompDistance := E_ErrorIdObjMgmt.ERRORID_InvalidCompressDistance;
END_IF
END_METHOD

METHOD M_SetCompFeed : ERRORID
VAR_INPUT
	nValue : DINT;
END_VAR
IF nValue >= cMinCompFeed AND nValue <= cMaxCompFeed THEN
	IF pFbFilamentExtruderRef > 0 THEN
		IF pFbFilamentExtruderRef^.P_nCompFeedOrgin <> nValue THEN
			pFbFilamentExtruderRef^.P_nCompFeedOrgin := nValue;
		END_IF
	END_IF
ELSE
	M_SetCompFeed := E_ErrorIdObjMgmt.ERRORID_InvalidCompressFeed;
END_IF
END_METHOD

METHOD M_SetDistance : ERRORID
VAR_INPUT
	nValue : DINT;
END_VAR
IF nValue >= cMinDistance AND nValue <= cMaxDistance THEN
	IF pFbFilamentExtruderRef > 0 THEN
		IF pFbFilamentExtruderRef^.P_nDistanceOrgin <> nValue THEN
			pFbFilamentExtruderRef^.P_nDistanceOrgin := nValue;
		END_IF
	END_IF
ELSE
	M_SetDistance := E_ErrorIdObjMgmt.ERRORID_InvalidExtrudeDistance;
END_IF
END_METHOD

METHOD M_SetFeed : ERRORID
VAR_INPUT
	nValue : DINT;
END_VAR
IF nValue >= cMinFeed AND nValue <= cMaxFeed THEN
	IF pFbFilamentExtruderRef > 0 THEN
		IF pFbFilamentExtruderRef^.P_nFeedOrgin <> nValue THEN
			pFbFilamentExtruderRef^.P_nFeedOrgin := nValue;
		END_IF
	END_IF
ELSE
	M_SetFeed := E_ErrorIdObjMgmt.ERRORID_InvalidExtrudeFeed;
END_IF
END_METHOD

METHOD M_SetRelaxDistance : ERRORID
VAR_INPUT
	nValue : DINT;
END_VAR
IF nValue >= cMinRelaxDistance AND nValue <= cMaxRelaxDistance THEN
	IF pFbFilamentExtruderRef > 0 THEN
		IF pFbFilamentExtruderRef^.P_nRelaxDistanceOrgin <> nValue THEN
			pFbFilamentExtruderRef^.P_nRelaxDistanceOrgin := nValue;
		END_IF
	END_IF
ELSE
	M_SetRelaxDistance := E_ErrorIdObjMgmt.ERRORID_InvalidRelaxDistance;
END_IF
END_METHOD

METHOD M_SetRelaxFeed : ERRORID
VAR_INPUT
	nValue : DINT;
END_VAR
IF nValue >= cMinRelaxFeed AND nValue <= cMaxRelaxFeed THEN
	IF pFbFilamentExtruderRef > 0 THEN
		IF pFbFilamentExtruderRef^.P_nRelaxFeedOrgin <> nValue THEN
			pFbFilamentExtruderRef^.P_nRelaxFeedOrgin := nValue;
		END_IF
	END_IF
ELSE
	M_SetRelaxFeed := E_ErrorIdObjMgmt.ERRORID_InvalidRelaxFeed;
END_IF
END_METHOD

METHOD M_StartStop
VAR_INPUT
	bStart : BOOL;
END_VAR
IF bStart AND NOT bBusy THEN
	bNormalStop := FALSE;
	bHardStop := FALSE;
	nState := 1;
ELSIF NOT bStart AND bBusy THEN
	bNormalStop := TRUE;
END_IF
END_METHOD

END_FUNCTION_BLOCK

// ---- Hardware/MultiZ/Extruder/FB_FDM_EL2521_Ref.TcPOU
FUNCTION_BLOCK FB_FDM_EL2521_Ref EXTENDS FB_ExtruderRef
VAR_INPUT
END_VAR
VAR
	pPTOStepperRef : POINTER TO ST_PTOStepperRef;
END_VAR
VAR_OUTPUT
	
END_VAR

